   1:  PR[GP1:91,2] = PR[GP1:90,2] + -16.413;
   1:L PR[91] R[100]mm/sec CNT100;
   1:  PR[GP1:91,1] = PR[GP1:90,1] + -9.727;
   1:  PR[GP1:91,2] = PR[GP1:90,2] + -15.652;
   1:L PR[91] R[100]mm/sec CNT100;
   1:  PR[GP1:91,1] = PR[GP1:90,1] + -6.729;
   1:  PR[GP1:91,2] = PR[GP1:90,2] + -12.994;
   1:L PR[91] R[100]mm/sec CNT100;
   1:  PR[GP1:91,1] = PR[GP1:90,1] + -6.347;
   1:  PR[GP1:91,2] = PR[GP1:90,2] + -12.598;
   1:L PR[91] R[100]mm/sec CNT100;
   1:  PR[GP1:91,1] = PR[GP1:90,1] + -4.072;
   1:  PR[GP1:91,2] = PR[GP1:90,2] + -9.212;
   1:L PR[91] R[100]mm/sec CNT100;
   1:  PR[GP1:91,1] = PR[GP1:90,1] + -3.579;
   1:  PR[GP1:91,2] = PR[GP1:90,2] + -8.510;
   1:L PR[91] R[100]mm/sec CNT100;
   1:  PR[GP1:91,1] = PR[GP1:90,1] + -3.207;
   1:  PR[GP1:91,2] = PR[GP1:90,2] + -8.109;
   1:L PR[91] R[100]mm/sec CNT100;
   1:  PR[GP1:91,1] = PR[GP1:90,1] + -2.834;
   1:  PR[GP1:91,2] = PR[GP1:90,2] + -7.762;
   1:L PR[91] R[100]mm/sec CNT100;
   1:  PR[GP1:91,1] = PR[GP1:90,1] + -2.234;
   1:  PR[GP1:91,2] = PR[GP1:90,2] + -7.336;
   1:L PR[91] R[100]mm/sec CNT100;
   1:  PR[GP1:91,1] = PR[GP1:90,1] + -1.110;
   1:  PR[GP1:91,2] = PR[GP1:90,2] + -7.075;
   1:L PR[91] R[100]mm/sec CNT100;
   1:  PR[GP1:91,1] = PR[GP1:90,1] + 1.269;
   1:L PR[91] R[100]mm/sec CNT100;
   1:  PR[GP1:91,1] = PR[GP1:90,1] + 2.391;
   1:  PR[GP1:91,2] = PR[GP1:90,2] + -7.335;
   1:L PR[91] R[100]mm/sec CNT100;
   1:  PR[GP1:91,1] = PR[GP1:90,1] + 2.990;
   1:  PR[GP1:91,2] = PR[GP1:90,2] + -7.760;
   1:L PR[91] R[100]mm/sec CNT100;
   1:  PR[GP1:91,1] = PR[GP1:90,1] + 3.095;
   1:  PR[GP1:91,2] = PR[GP1:90,2] + -7.857;
   1:L PR[91] R[100]mm/sec CNT100;
   1:  PR[GP1:91,1] = PR[GP1:90,1] + 3.258;
   1:  PR[GP1:91,2] = PR[GP1:90,2] + -7.827;
   1:L PR[91] R[100]mm/sec CNT100;
   1:  PR[GP1:91,1] = PR[GP1:90,1] + 4.180;
   1:  PR[GP1:91,2] = PR[GP1:90,2] + -9.139;
   1:L PR[91] R[100]mm/sec CNT100;
   1:  PR[GP1:91,1] = PR[GP1:90,1] + 6.503;
   1:  PR[GP1:91,2] = PR[GP1:90,2] + -12.593;
   1:L PR[91] R[100]mm/sec CNT100;
   1:  PR[GP1:91,1] = PR[GP1:90,1] + 6.887;
   1:  PR[GP1:91,2] = PR[GP1:90,2] + -12.991;
   1:L PR[91] R[100]mm/sec CNT100;
   1:  PR[GP1:91,1] = PR[GP1:90,1] + 9.883;
   1:  PR[GP1:91,2] = PR[GP1:90,2] + -15.654;
   1:L PR[91] R[100]mm/sec CNT100;
   1:  PR[GP1:91,1] = PR[GP1:90,1] + 11.125;
   1:  PR[GP1:91,2] = PR[GP1:90,2] + -16.415;
   1:L PR[91] R[100]mm/sec CNT100;
   1:  PR[GP1:91,1] = PR[GP1:90,1] + 13.931;
   1:  PR[GP1:91,2] = PR[GP1:90,2] + -17.885;
   1:L PR[91] R[100]mm/sec CNT100;
   1:  PR[GP1:91,1] = PR[GP1:90,1] + 16.261;
   1:  PR[GP1:91,2] = PR[GP1:90,2] + -18.611;
   1:L PR[91] R[100]mm/sec CNT100;
   1:  PR[GP1:91,1] = PR[GP1:90,1] + 18.451;
   1:  PR[GP1:91,2] = PR[GP1:90,2] + -19.161;
   1:L PR[91] R[100]mm/sec CNT100;
   1:  PR[GP1:91,1] = PR[GP1:90,1] + 21.839;
   1:  PR[GP1:91,2] = PR[GP1:90,2] + -19.352;
   1:L PR[91] R[100]mm/sec CNT100;
   1:  PR[GP1:91,1] = PR[GP1:90,1] + 23.204;
   1:  PR[GP1:91,2] = PR[GP1:90,2] + -19.363;
   1:L PR[91] R[100]mm/sec CNT100;
   1:  PR[GP1:91,1] = PR[GP1:90,1] + 27.366;
   1:  PR[GP1:91,2] = PR[GP1:90,2] + -18.570;
   1:L PR[91] R[100]mm/sec CNT100;
   1:  PR[GP1:91,1] = PR[GP1:90,1] + 27.918;
   1:  PR[GP1:91,2] = PR[GP1:90,2] + -18.441;
   1:L PR[91] R[100]mm/sec CNT100;
   1:  PR[GP1:91,1] = PR[GP1:90,1] + 32.318;
   1:  PR[GP1:91,2] = PR[GP1:90,2] + -16.403;
   1:L PR[91] R[100]mm/sec CNT100;
   1:  PR[GP1:91,1] = PR[GP1:90,1] + 36.034;
   1:  PR[GP1:91,2] = PR[GP1:90,2] + -13.380;
   1:L PR[91] R[100]mm/sec CNT100;
   1:  PR[GP1:91,1] = PR[GP1:90,1] + 38.885;
   1:  PR[GP1:91,2] = PR[GP1:90,2] + -9.507;
   1:L PR[91] R[100]mm/sec CNT100;
   1:  PR[GP1:91,1] = PR[GP1:90,1] + 40.679;
   1:  PR[GP1:91,2] = PR[GP1:90,2] + -5.092;
   1:L PR[91] R[100]mm/sec CNT100;
   1:  PR[GP1:91,1] = PR[GP1:90,1] + 40.772;
   1:  PR[GP1:91,2] = PR[GP1:90,2] + -4.390;
   1:L PR[91] R[100]mm/sec CNT100;
   1:  PR[GP1:91,1] = PR[GP1:90,1] + 41.290;
   1:  PR[GP1:91,2] = PR[GP1:90,2] + -0.313;
   1:L PR[91] R[100]mm/sec CNT100;
   1:  PR[GP1:91,1] = PR[GP1:90,1] + 40.677;
   1:  PR[GP1:91,2] = PR[GP1:90,2] + 4.471;
   1:L PR[91] R[100]mm/sec CNT100;
   1:  PR[GP1:91,1] = PR[GP1:90,1] + 38.885;
   1:  PR[GP1:91,2] = PR[GP1:90,2] + 8.882;
   1:L PR[91] R[100]mm/sec CNT100;
   1:  PR[GP1:91,1] = PR[GP1:90,1] + 36.035;
   1:  PR[GP1:91,2] = PR[GP1:90,2] + 12.755;
   1:L PR[91] R[100]mm/sec CNT100;
   1:  PR[GP1:91,1] = PR[GP1:90,1] + 32.320;
   1:  PR[GP1:91,2] = PR[GP1:90,2] + 15.778;
   1:L PR[91] R[100]mm/sec CNT100;
   1:  PR[GP1:91,1] = PR[GP1:90,1] + 27.921;
   1:  PR[GP1:91,2] = PR[GP1:90,2] + 17.816;
   1:L PR[91] R[100]mm/sec CNT100;
   1:  PR[GP1:91,1] = PR[GP1:90,1] + 27.368;
   1:  PR[GP1:91,2] = PR[GP1:90,2] + 17.945;
   1:L PR[91] R[100]mm/sec CNT100;
   1:  PR[GP1:91,1] = PR[GP1:90,1] + 23.206;
   1:  PR[GP1:91,2] = PR[GP1:90,2] + 18.739;
   1:L PR[91] R[100]mm/sec CNT100;
   1:  PR[GP1:91,1] = PR[GP1:90,1] + 21.839;
   1:  PR[GP1:91,2] = PR[GP1:90,2] + 18.728;
   1:L PR[91] R[100]mm/sec CNT100;
   1:  PR[GP1:91,1] = PR[GP1:90,1] + 18.450;
   1:  PR[GP1:91,2] = PR[GP1:90,2] + 18.537;
   1:L PR[91] R[100]mm/sec CNT100;
   1:  PR[GP1:91,1] = PR[GP1:90,1] + 16.257;
   1:  PR[GP1:91,2] = PR[GP1:90,2] + 17.986;
   1:L PR[91] R[100]mm/sec CNT100;
   1:  PR[GP1:91,1] = PR[GP1:90,1] + 13.927;
   1:  PR[GP1:91,2] = PR[GP1:90,2] + 17.260;
   1:L PR[91] R[100]mm/sec CNT100;
   1:  PR[GP1:91,1] = PR[GP1:90,1] + 11.119;
   1:  PR[GP1:91,2] = PR[GP1:90,2] + 15.786;
   1:L PR[91] R[100]mm/sec CNT100;
   1:  PR[GP1:91,1] = PR[GP1:90,1] + 9.878;
   1:  PR[GP1:91,2] = PR[GP1:90,2] + 15.026;
   1:L PR[91] R[100]mm/sec CNT100;
   1:  PR[GP1:91,1] = PR[GP1:90,1] + 6.878;
   1:  PR[GP1:91,2] = PR[GP1:90,2] + 12.357;
   1:L PR[91] R[100]mm/sec CNT100;
   1:  PR[GP1:91,1] = PR[GP1:90,1] + 6.495;
   1:  PR[GP1:91,2] = PR[GP1:90,2] + 11.959;
   1:L PR[91] R[100]mm/sec CNT100;
   1:  PR[GP1:91,1] = PR[GP1:90,1] + 3.744;
   1:  PR[GP1:91,2] = PR[GP1:90,2] + 7.889;
   1:L PR[91] R[100]mm/sec CNT100;
   1:  PR[GP1:91,1] = PR[GP1:90,1] + 3.363;
   1:  PR[GP1:91,2] = PR[GP1:90,2] + 7.482;
   1:L PR[91] R[100]mm/sec CNT100;
   1:  PR[GP1:91,1] = PR[GP1:90,1] + 2.992;
   1:  PR[GP1:91,2] = PR[GP1:90,2] + 7.138;
   1:L PR[91] R[100]mm/sec CNT100;
   1:  PR[GP1:91,1] = PR[GP1:90,1] + 2.394;
   1:  PR[GP1:91,2] = PR[GP1:90,2] + 6.712;
   1:L PR[91] R[100]mm/sec CNT100;
   1:  PR[GP1:91,1] = PR[GP1:90,1] + 1.274;
   1:  PR[GP1:91,2] = PR[GP1:90,2] + 6.451;
   1:L PR[91] R[100]mm/sec CNT100;
   1:  PR[GP1:91,1] = PR[GP1:90,1] + -1.109;
   1:L PR[91] R[100]mm/sec CNT100;
   1:  ! -- Layer/Ebene 29 -- !;
   1:  PR[91] = PR[90];
   1:  PR[GP1:91,1] = PR[GP1:90,1] + -2.164;
   1:  PR[GP1:91,2] = PR[GP1:90,2] + 7.007;
   1:  PR[GP1:91,3] = PR[GP1:90,3] + 17.995;
   1:L PR[91] R[100]mm/sec CNT100;
   1:  PR[GP1:91,1] = PR[GP1:90,1] + -2.721;
   1:  PR[GP1:91,2] = PR[GP1:90,2] + 7.403;
   1:L PR[91] R[100]mm/sec CNT100;
   1:  PR[GP1:91,1] = PR[GP1:90,1] + -3.141;
   1:  PR[GP1:91,2] = PR[GP1:90,2] + 7.794;
   1:L PR[91] R[100]mm/sec CNT100;
   1:  PR[GP1:91,1] = PR[GP1:90,1] + -3.471;
   1:  PR[GP1:91,2] = PR[GP1:90,2] + 8.153;
   1:L PR[91] R[100]mm/sec CNT100;
   1:  PR[GP1:91,1] = PR[GP1:90,1] + -6.256;
   1:  PR[GP1:91,2] = PR[GP1:90,2] + 12.114;
   1:L PR[91] R[100]mm/sec CNT100;
   1:  PR[GP1:91,1] = PR[GP1:90,1] + -9.715;
   1:  PR[GP1:91,2] = PR[GP1:90,2] + 15.175;
   1:L PR[91] R[100]mm/sec CNT100;
   1:  PR[GP1:91,1] = PR[GP1:90,1] + -10.311;
   1:  PR[GP1:91,2] = PR[GP1:90,2] + 15.540;
   1:L PR[91] R[100]mm/sec CNT100;
   1:  PR[GP1:91,1] = PR[GP1:90,1] + -13.770;
   1:  PR[GP1:91,2] = PR[GP1:90,2] + 17.357;
   1:L PR[91] R[100]mm/sec CNT100;
   1:  PR[GP1:91,1] = PR[GP1:90,1] + -15.408;
   1:  PR[GP1:91,2] = PR[GP1:90,2] + 17.867;
   1:L PR[91] R[100]mm/sec CNT100;
   1:  PR[GP1:91,1] = PR[GP1:90,1] + -18.283;
   1:  PR[GP1:91,2] = PR[GP1:90,2] + 18.587;
   1:L PR[91] R[100]mm/sec CNT100;
   1:  PR[GP1:91,1] = PR[GP1:90,1] + -20.988;
   1:  PR[GP1:91,2] = PR[GP1:90,2] + 18.739;
   1:L PR[91] R[100]mm/sec CNT100;
   1:  PR[GP1:91,1] = PR[GP1:90,1] + -23.021;
   1:  PR[GP1:91,2] = PR[GP1:90,2] + 18.755;
   1:L PR[91] R[100]mm/sec CNT100;
   1:  PR[GP1:91,1] = PR[GP1:90,1] + -26.552;
   1:  PR[GP1:91,2] = PR[GP1:90,2] + 18.083;
   1:L PR[91] R[100]mm/sec CNT100;
   1:  PR[GP1:91,1] = PR[GP1:90,1] + -27.715;
   1:  PR[GP1:91,2] = PR[GP1:90,2] + 17.812;
   1:L PR[91] R[100]mm/sec CNT100;
   1:  PR[GP1:91,1] = PR[GP1:90,1] + -31.631;
   1:  PR[GP1:91,2] = PR[GP1:90,2] + 15.998;
   1:L PR[91] R[100]mm/sec CNT100;
   1:  PR[GP1:91,1] = PR[GP1:90,1] + -32.075;
   1:  PR[GP1:91,2] = PR[GP1:90,2] + 15.774;
   1:L PR[91] R[100]mm/sec CNT100;
   1:  PR[GP1:91,1] = PR[GP1:90,1] + -35.827;
   1:  PR[GP1:91,2] = PR[GP1:90,2] + 12.731;
   1:L PR[91] R[100]mm/sec CNT100;
   1:  PR[GP1:91,1] = PR[GP1:90,1] + -38.675;
   1:  PR[GP1:91,2] = PR[GP1:90,2] + 8.865;
   1:L PR[91] R[100]mm/sec CNT100;
   1:  PR[GP1:91,1] = PR[GP1:90,1] + -40.458;
   1:  PR[GP1:91,2] = PR[GP1:90,2] + 4.452;
   1:L PR[91] R[100]mm/sec CNT100;
   1:  PR[GP1:91,1] = PR[GP1:90,1] + -41.066;
   1:  PR[GP1:91,2] = PR[GP1:90,2] + -0.312;
   1:L PR[91] R[100]mm/sec CNT100;
   1:  PR[GP1:91,1] = PR[GP1:90,1] + -40.458;
   1:  PR[GP1:91,2] = PR[GP1:90,2] + -5.076;
   1:L PR[91] R[100]mm/sec CNT100;
   1:  PR[GP1:91,1] = PR[GP1:90,1] + -38.674;
   1:  PR[GP1:91,2] = PR[GP1:90,2] + -9.491;
   1:L PR[91] R[100]mm/sec CNT100;
   1:  PR[GP1:91,1] = PR[GP1:90,1] + -36.976;
   1:  PR[GP1:91,2] = PR[GP1:90,2] + -11.803;
   1:L PR[91] R[100]mm/sec CNT100;
   1:  PR[GP1:91,1] = PR[GP1:90,1] + -35.828;
   1:  PR[GP1:91,2] = PR[GP1:90,2] + -13.354;
   1:L PR[91] R[100]mm/sec CNT100;
   1:  PR[GP1:91,1] = PR[GP1:90,1] + -32.074;
   1:  PR[GP1:91,2] = PR[GP1:90,2] + -16.398;
   1:L PR[91] R[100]mm/sec CNT100;
   1:  PR[GP1:91,1] = PR[GP1:90,1] + -31.630;
   1:  PR[GP1:91,2] = PR[GP1:90,2] + -16.622;
   1:L PR[91] R[100]mm/sec CNT100;
   1:  PR[GP1:91,1] = PR[GP1:90,1] + -27.714;
   1:  PR[GP1:91,2] = PR[GP1:90,2] + -18.436;
   1:L PR[91] R[100]mm/sec CNT100;
   1:  PR[GP1:91,1] = PR[GP1:90,1] + -26.551;
   1:  PR[GP1:91,2] = PR[GP1:90,2] + -18.707;
   1:L PR[91] R[100]mm/sec CNT100;
   1:  PR[GP1:91,1] = PR[GP1:90,1] + -23.020;
   1:  PR[GP1:91,2] = PR[GP1:90,2] + -19.379;
   1:L PR[91] R[100]mm/sec CNT100;
   1:  PR[GP1:91,1] = PR[GP1:90,1] + -20.987;
   1:  PR[GP1:91,2] = PR[GP1:90,2] + -19.363;
   1:L PR[91] R[100]mm/sec CNT100;
   1:  PR[GP1:91,1] = PR[GP1:90,1] + -18.282;
   1:  PR[GP1:91,2] = PR[GP1:90,2] + -19.210;
   1:L PR[91] R[100]mm/sec CNT100;
   1:  PR[GP1:91,1] = PR[GP1:90,1] + -15.407;
   1:  PR[GP1:91,2] = PR[GP1:90,2] + -18.491;
   1:L PR[91] R[100]mm/sec CNT100;
   1:  PR[GP1:91,1] = PR[GP1:90,1] + -13.770;
   1:  PR[GP1:91,2] = PR[GP1:90,2] + -17.981;
   1:L PR[91] R[100]mm/sec CNT100;
   1:  PR[GP1:91,1] = PR[GP1:90,1] + -10.310;
   1:  PR[GP1:91,2] = PR[GP1:90,2] + -16.164;
   1:L PR[91] R[100]mm/sec CNT100;
   1:  PR[GP1:91,1] = PR[GP1:90,1] + -9.714;
   1:  PR[GP1:91,2] = PR[GP1:90,2] + -15.798;
   1:L PR[91] R[100]mm/sec CNT100;
   1:  PR[GP1:91,1] = PR[GP1:90,1] + -6.255;
   1:  PR[GP1:91,2] = PR[GP1:90,2] + -12.737;
   1:L PR[91] R[100]mm/sec CNT100;
   1:  PR[GP1:91,1] = PR[GP1:90,1] + -3.471;
   1:  PR[GP1:91,2] = PR[GP1:90,2] + -8.774;
   1:L PR[91] R[100]mm/sec CNT100;
   1:  PR[GP1:91,1] = PR[GP1:90,1] + -3.139;
   1:  PR[GP1:91,2] = PR[GP1:90,2] + -8.415;
   1:L PR[91] R[100]mm/sec CNT100;
   1:  PR[GP1:91,1] = PR[GP1:90,1] + -2.720;
   1:  PR[GP1:91,2] = PR[GP1:90,2] + -8.026;
   1:L PR[91] R[100]mm/sec CNT100;
   1:  PR[GP1:91,1] = PR[GP1:90,1] + -2.163;
   1:  PR[GP1:91,2] = PR[GP1:90,2] + -7.630;
   1:L PR[91] R[100]mm/sec CNT100;
   1:  PR[GP1:91,1] = PR[GP1:90,1] + -1.030;
   1:  PR[GP1:91,2] = PR[GP1:90,2] + -7.363;
   1:L PR[91] R[100]mm/sec CNT100;
   1:  PR[GP1:91,1] = PR[GP1:90,1] + 1.190;
   1:L PR[91] R[100]mm/sec CNT100;
   1:  PR[GP1:91,1] = PR[GP1:90,1] + 2.321;
   1:  PR[GP1:91,2] = PR[GP1:90,2] + -7.630;
   1:L PR[91] R[100]mm/sec CNT100;
   1:  PR[GP1:91,1] = PR[GP1:90,1] + 2.877;
   1:  PR[GP1:91,2] = PR[GP1:90,2] + -8.024;
   1:L PR[91] R[100]mm/sec CNT100;
   1:  PR[GP1:91,1] = PR[GP1:90,1] + 2.984;
   1:  PR[GP1:91,2] = PR[GP1:90,2] + -8.123;
   1:L PR[91] R[100]mm/sec CNT100;
   1:  PR[GP1:91,1] = PR[GP1:90,1] + 3.151;
   1:  PR[GP1:91,2] = PR[GP1:90,2] + -8.091;
   1:L PR[91] R[100]mm/sec CNT100;
   1:  PR[GP1:91,1] = PR[GP1:90,1] + 6.413;
   1:  PR[GP1:91,2] = PR[GP1:90,2] + -12.733;
   1:L PR[91] R[100]mm/sec CNT100;
   1:  PR[GP1:91,1] = PR[GP1:90,1] + 9.871;
   1:  PR[GP1:91,2] = PR[GP1:90,2] + -15.802;
   1:L PR[91] R[100]mm/sec CNT100;
   1:  PR[GP1:91,1] = PR[GP1:90,1] + 10.466;
   1:  PR[GP1:91,2] = PR[GP1:90,2] + -16.166;
   1:L PR[91] R[100]mm/sec CNT100;
   1:  PR[GP1:91,1] = PR[GP1:90,1] + 13.925;
   1:  PR[GP1:91,2] = PR[GP1:90,2] + -17.979;
   1:L PR[91] R[100]mm/sec CNT100;
   1:  PR[GP1:91,1] = PR[GP1:90,1] + 15.563;
   1:  PR[GP1:91,2] = PR[GP1:90,2] + -18.490;
   1:L PR[91] R[100]mm/sec CNT100;
   1:  PR[GP1:91,1] = PR[GP1:90,1] + 18.437;
   1:  PR[GP1:91,2] = PR[GP1:90,2] + -19.210;
   1:L PR[91] R[100]mm/sec CNT100;
   1:  PR[GP1:91,1] = PR[GP1:90,1] + 21.142;
   1:  PR[GP1:91,2] = PR[GP1:90,2] + -19.363;
   1:L PR[91] R[100]mm/sec CNT100;
   1:  PR[GP1:91,1] = PR[GP1:90,1] + 23.175;
   1:  PR[GP1:91,2] = PR[GP1:90,2] + -19.380;
   1:L PR[91] R[100]mm/sec CNT100;
   1:  PR[GP1:91,1] = PR[GP1:90,1] + 26.706;
   1:  PR[GP1:91,2] = PR[GP1:90,2] + -18.707;
   1:L PR[91] R[100]mm/sec CNT100;
   1:  PR[GP1:91,1] = PR[GP1:90,1] + 27.869;
   1:  PR[GP1:91,2] = PR[GP1:90,2] + -18.435;
   1:L PR[91] R[100]mm/sec CNT100;
   1:  PR[GP1:91,1] = PR[GP1:90,1] + 31.786;
   1:  PR[GP1:91,2] = PR[GP1:90,2] + -16.624;
   1:L PR[91] R[100]mm/sec CNT100;
   1:  PR[GP1:91,1] = PR[GP1:90,1] + 32.230;
   1:  PR[GP1:91,2] = PR[GP1:90,2] + -16.401;
   1:L PR[91] R[100]mm/sec CNT100;
   1:  PR[GP1:91,1] = PR[GP1:90,1] + 35.973;
   1:  PR[GP1:91,2] = PR[GP1:90,2] + -13.368;
   1:L PR[91] R[100]mm/sec CNT100;
   1:  PR[GP1:91,1] = PR[GP1:90,1] + 38.831;
   1:  PR[GP1:91,2] = PR[GP1:90,2] + -9.486;
   1:L PR[91] R[100]mm/sec CNT100;
   1:  PR[GP1:91,1] = PR[GP1:90,1] + 40.616;
   1:  PR[GP1:91,2] = PR[GP1:90,2] + -5.083;
   1:L PR[91] R[100]mm/sec CNT100;
   1:  PR[GP1:91,1] = PR[GP1:90,1] + 40.644;
   1:  PR[GP1:91,2] = PR[GP1:90,2] + -4.869;
   1:L PR[91] R[100]mm/sec CNT100;
   1:  PR[GP1:91,1] = PR[GP1:90,1] + 41.223;
   1:  PR[GP1:91,2] = PR[GP1:90,2] + -0.312;
   1:L PR[91] R[100]mm/sec CNT100;
   1:  PR[GP1:91,1] = PR[GP1:90,1] + 40.615;
   1:  PR[GP1:91,2] = PR[GP1:90,2] + 4.462;
   1:L PR[91] R[100]mm/sec CNT100;
   1:  PR[GP1:91,1] = PR[GP1:90,1] + 38.832;
   1:  PR[GP1:91,2] = PR[GP1:90,2] + 8.861;
   1:L PR[91] R[100]mm/sec CNT100;
   1:  PR[GP1:91,1] = PR[GP1:90,1] + 35.983;
   1:  PR[GP1:91,2] = PR[GP1:90,2] + 12.731;
   1:L PR[91] R[100]mm/sec CNT100;
   1:  PR[GP1:91,1] = PR[GP1:90,1] + 32.232;
   1:  PR[GP1:91,2] = PR[GP1:90,2] + 15.776;
   1:L PR[91] R[100]mm/sec CNT100;
   1:  PR[GP1:91,1] = PR[GP1:90,1] + 31.788;
   1:  PR[GP1:91,2] = PR[GP1:90,2] + 15.999;
   1:L PR[91] R[100]mm/sec CNT100;
   1:  PR[GP1:91,1] = PR[GP1:90,1] + 27.870;
   1:  PR[GP1:91,2] = PR[GP1:90,2] + 17.811;
   1:L PR[91] R[100]mm/sec CNT100;
   1:  PR[GP1:91,1] = PR[GP1:90,1] + 26.706;
   1:  PR[GP1:91,2] = PR[GP1:90,2] + 18.082;
   1:L PR[91] R[100]mm/sec CNT100;
   1:  PR[GP1:91,1] = PR[GP1:90,1] + 23.175;
   1:  PR[GP1:91,2] = PR[GP1:90,2] + 18.756;
   1:L PR[91] R[100]mm/sec CNT100;
   1:  PR[GP1:91,1] = PR[GP1:90,1] + 21.139;
   1:  PR[GP1:91,2] = PR[GP1:90,2] + 18.738;
   1:L PR[91] R[100]mm/sec CNT100;
   1:  PR[GP1:91,1] = PR[GP1:90,1] + 18.435;
   1:  PR[GP1:91,2] = PR[GP1:90,2] + 18.586;
   1:L PR[91] R[100]mm/sec CNT100;
   1:  PR[GP1:91,1] = PR[GP1:90,1] + 15.557;
   1:  PR[GP1:91,2] = PR[GP1:90,2] + 17.863;
   1:L PR[91] R[100]mm/sec CNT100;
   1:  PR[GP1:91,1] = PR[GP1:90,1] + 13.919;
   1:  PR[GP1:91,2] = PR[GP1:90,2] + 17.353;
   1:L PR[91] R[100]mm/sec CNT100;
   1:  PR[GP1:91,1] = PR[GP1:90,1] + 10.457;
   1:  PR[GP1:91,2] = PR[GP1:90,2] + 15.535;
   1:L PR[91] R[100]mm/sec CNT100;
   1:  PR[GP1:91,1] = PR[GP1:90,1] + 9.863;
   1:  PR[GP1:91,2] = PR[GP1:90,2] + 15.172;
   1:L PR[91] R[100]mm/sec CNT100;
   1:  PR[GP1:91,1] = PR[GP1:90,1] + 6.404;
   1:  PR[GP1:91,2] = PR[GP1:90,2] + 12.099;
   1:L PR[91] R[100]mm/sec CNT100;
   1:  PR[GP1:91,1] = PR[GP1:90,1] + 3.629;
   1:  PR[GP1:91,2] = PR[GP1:90,2] + 8.144;
   1:L PR[91] R[100]mm/sec CNT100;
   1:  PR[GP1:91,1] = PR[GP1:90,1] + 3.295;
   1:  PR[GP1:91,2] = PR[GP1:90,2] + 7.788;
   1:L PR[91] R[100]mm/sec CNT100;
   1:  PR[GP1:91,1] = PR[GP1:90,1] + 2.879;
   1:  PR[GP1:91,2] = PR[GP1:90,2] + 7.402;
   1:L PR[91] R[100]mm/sec CNT100;
   1:  PR[GP1:91,1] = PR[GP1:90,1] + 2.324;
   1:  PR[GP1:91,2] = PR[GP1:90,2] + 7.007;
   1:L PR[91] R[100]mm/sec CNT100;
   1:  PR[GP1:91,1] = PR[GP1:90,1] + 1.195;
   1:  PR[GP1:91,2] = PR[GP1:90,2] + 6.739;
   1:L PR[91] R[100]mm/sec CNT100;
   1:  PR[GP1:91,1] = PR[GP1:90,1] + -1.030;
   1:L PR[91] R[100]mm/sec CNT100;
   1:  ! -- Layer/Ebene 30 -- !;
   1:  PR[91] = PR[90];
   1:  PR[GP1:91,1] = PR[GP1:90,1] + -2.093;
   1:  PR[GP1:91,2] = PR[GP1:90,2] + 7.301;
   1:  PR[GP1:91,3] = PR[GP1:90,3] + 18.605;
   1:L PR[91] R[100]mm/sec CNT100;
   1:  PR[GP1:91,1] = PR[GP1:90,1] + -2.607;
   1:  PR[GP1:91,2] = PR[GP1:90,2] + 7.667;
   1:L PR[91] R[100]mm/sec CNT100;
   1:  PR[GP1:91,1] = PR[GP1:90,1] + -3.073;
   1:  PR[GP1:91,2] = PR[GP1:90,2] + 8.100;
   1:L PR[91] R[100]mm/sec CNT100;
   1:  PR[GP1:91,1] = PR[GP1:90,1] + -3.365;
   1:  PR[GP1:91,2] = PR[GP1:90,2] + 8.417;
   1:L PR[91] R[100]mm/sec CNT100;
   1:  PR[GP1:91,1] = PR[GP1:90,1] + -5.728;
   1:  PR[GP1:91,2] = PR[GP1:90,2] + 11.782;
   1:L PR[91] R[100]mm/sec CNT100;
   1:  PR[GP1:91,1] = PR[GP1:90,1] + -5.998;
   1:  PR[GP1:91,2] = PR[GP1:90,2] + 12.131;
   1:L PR[91] R[100]mm/sec CNT100;
   1:  PR[GP1:91,1] = PR[GP1:90,1] + -9.684;
   1:  PR[GP1:91,2] = PR[GP1:90,2] + 15.308;
   1:L PR[91] R[100]mm/sec CNT100;
   1:  PR[GP1:91,1] = PR[GP1:90,1] + -13.764;
   1:  PR[GP1:91,2] = PR[GP1:90,2] + 17.451;
   1:L PR[91] R[100]mm/sec CNT100;
   1:  PR[GP1:91,1] = PR[GP1:90,1] + -14.709;
   1:  PR[GP1:91,2] = PR[GP1:90,2] + 17.746;
   1:L PR[91] R[100]mm/sec CNT100;
   1:  PR[GP1:91,1] = PR[GP1:90,1] + -18.269;
   1:  PR[GP1:91,2] = PR[GP1:90,2] + 18.636;
   1:L PR[91] R[100]mm/sec CNT100;
   1:  PR[GP1:91,1] = PR[GP1:90,1] + -20.290;
   1:  PR[GP1:91,2] = PR[GP1:90,2] + 18.750;
   1:L PR[91] R[100]mm/sec CNT100;
   1:  PR[GP1:91,1] = PR[GP1:90,1] + -22.991;
   1:  PR[GP1:91,2] = PR[GP1:90,2] + 18.772;
   1:L PR[91] R[100]mm/sec CNT100;
   1:  PR[GP1:91,1] = PR[GP1:90,1] + -25.892;
   1:  PR[GP1:91,2] = PR[GP1:90,2] + 18.219;
   1:L PR[91] R[100]mm/sec CNT100;
   1:  PR[GP1:91,1] = PR[GP1:90,1] + -27.664;
   1:  PR[GP1:91,2] = PR[GP1:90,2] + 17.807;
   1:L PR[91] R[100]mm/sec CNT100;
   1:  PR[GP1:91,1] = PR[GP1:90,1] + -31.036;
   1:  PR[GP1:91,2] = PR[GP1:90,2] + 16.244;
   1:L PR[91] R[100]mm/sec CNT100;
   1:  PR[GP1:91,1] = PR[GP1:90,1] + -32.004;
   1:  PR[GP1:91,2] = PR[GP1:90,2] + 15.757;
   1:L PR[91] R[100]mm/sec CNT100;
   1:  PR[GP1:91,1] = PR[GP1:90,1] + -35.336;
   1:  PR[GP1:91,2] = PR[GP1:90,2] + 13.058;
   1:L PR[91] R[100]mm/sec CNT100;
   1:  PR[GP1:91,1] = PR[GP1:90,1] + -35.728;
   1:  PR[GP1:91,2] = PR[GP1:90,2] + 12.724;
   1:L PR[91] R[100]mm/sec CNT100;
   1:  PR[GP1:91,1] = PR[GP1:90,1] + -38.512;
   1:  PR[GP1:91,2] = PR[GP1:90,2] + 8.963;
   1:L PR[91] R[100]mm/sec CNT100;
   1:  PR[GP1:91,1] = PR[GP1:90,1] + -38.587;
   1:  PR[GP1:91,2] = PR[GP1:90,2] + 8.857;
   1:L PR[91] R[100]mm/sec CNT100;
   1:  PR[GP1:91,1] = PR[GP1:90,1] + -40.387;
   1:  PR[GP1:91,2] = PR[GP1:90,2] + 4.439;
   1:L PR[91] R[100]mm/sec CNT100;
   1:  PR[GP1:91,1] = PR[GP1:90,1] + -41.000;
   1:  PR[GP1:91,2] = PR[GP1:90,2] + -0.312;
   1:L PR[91] R[100]mm/sec CNT100;
   1:  PR[GP1:91,1] = PR[GP1:90,1] + -40.387;
   1:  PR[GP1:91,2] = PR[GP1:90,2] + -5.063;
   1:L PR[91] R[100]mm/sec CNT100;
   1:  PR[GP1:91,1] = PR[GP1:90,1] + -38.592;
   1:  PR[GP1:91,2] = PR[GP1:90,2] + -9.468;
   1:L PR[91] R[100]mm/sec CNT100;
   1:  PR[GP1:91,1] = PR[GP1:90,1] + -35.727;
   1:  PR[GP1:91,2] = PR[GP1:90,2] + -13.349;
   1:L PR[91] R[100]mm/sec CNT100;
   1:  PR[GP1:91,1] = PR[GP1:90,1] + -35.335;
   1:  PR[GP1:91,2] = PR[GP1:90,2] + -13.683;
   1:L PR[91] R[100]mm/sec CNT100;
   1:  PR[GP1:91,1] = PR[GP1:90,1] + -32.004;
   1:  PR[GP1:91,2] = PR[GP1:90,2] + -16.381;
   1:L PR[91] R[100]mm/sec CNT100;
   1:  PR[GP1:91,1] = PR[GP1:90,1] + -31.036;
   1:  PR[GP1:91,2] = PR[GP1:90,2] + -16.869;
   1:L PR[91] R[100]mm/sec CNT100;
   1:  PR[GP1:91,1] = PR[GP1:90,1] + -27.664;
   1:  PR[GP1:91,2] = PR[GP1:90,2] + -18.431;
   1:L PR[91] R[100]mm/sec CNT100;
   1:  PR[GP1:91,1] = PR[GP1:90,1] + -25.891;
   1:  PR[GP1:91,2] = PR[GP1:90,2] + -18.843;
   1:L PR[91] R[100]mm/sec CNT100;
   1:  PR[GP1:91,1] = PR[GP1:90,1] + -22.990;
   1:  PR[GP1:91,2] = PR[GP1:90,2] + -19.396;
   1:L PR[91] R[100]mm/sec CNT100;
   1:  PR[GP1:91,1] = PR[GP1:90,1] + -20.289;
   1:  PR[GP1:91,2] = PR[GP1:90,2] + -19.374;
   1:L PR[91] R[100]mm/sec CNT100;
   1:  PR[GP1:91,1] = PR[GP1:90,1] + -18.268;
   1:  PR[GP1:91,2] = PR[GP1:90,2] + -19.260;
   1:L PR[91] R[100]mm/sec CNT100;
   1:  PR[GP1:91,1] = PR[GP1:90,1] + -14.708;
   1:  PR[GP1:91,2] = PR[GP1:90,2] + -18.369;
   1:L PR[91] R[100]mm/sec CNT100;
   1:  PR[GP1:91,1] = PR[GP1:90,1] + -13.763;
   1:  PR[GP1:91,2] = PR[GP1:90,2] + -18.075;
   1:L PR[91] R[100]mm/sec CNT100;
   1:  PR[GP1:91,1] = PR[GP1:90,1] + -9.690;
   1:  PR[GP1:91,2] = PR[GP1:90,2] + -15.935;
   1:L PR[91] R[100]mm/sec CNT100;
   1:  PR[GP1:91,1] = PR[GP1:90,1] + -9.338;
   1:  PR[GP1:91,2] = PR[GP1:90,2] + -15.623;
   1:L PR[91] R[100]mm/sec CNT100;
   1:  PR[GP1:91,1] = PR[GP1:90,1] + -6.247;
   1:  PR[GP1:91,2] = PR[GP1:90,2] + -12.988;
   1:L PR[91] R[100]mm/sec CNT100;
   1:  PR[GP1:91,1] = PR[GP1:90,1] + -6.011;
   1:  PR[GP1:91,2] = PR[GP1:90,2] + -12.772;
   1:L PR[91] R[100]mm/sec CNT100;
   1:  PR[GP1:91,1] = PR[GP1:90,1] + -5.728;
   1:  PR[GP1:91,2] = PR[GP1:90,2] + -12.406;
   1:L PR[91] R[100]mm/sec CNT100;
   1:  PR[GP1:91,1] = PR[GP1:90,1] + -3.364;
   1:  PR[GP1:91,2] = PR[GP1:90,2] + -9.038;
   1:L PR[91] R[100]mm/sec CNT100;
   1:  PR[GP1:91,1] = PR[GP1:90,1] + -3.070;
   1:  PR[GP1:91,2] = PR[GP1:90,2] + -8.722;
   1:L PR[91] R[100]mm/sec CNT100;
   1:  PR[GP1:91,1] = PR[GP1:90,1] + -2.607;
   1:  PR[GP1:91,2] = PR[GP1:90,2] + -8.291;
   1:L PR[91] R[100]mm/sec CNT100;
   1:  PR[GP1:91,1] = PR[GP1:90,1] + -2.093;
   1:  PR[GP1:91,2] = PR[GP1:90,2] + -7.925;
   1:L PR[91] R[100]mm/sec CNT100;
   1:  PR[GP1:91,1] = PR[GP1:90,1] + -0.950;
   1:  PR[GP1:91,2] = PR[GP1:90,2] + -7.652;
   1:L PR[91] R[100]mm/sec CNT100;
   1:  PR[GP1:91,1] = PR[GP1:90,1] + 1.111;
   1:L PR[91] R[100]mm/sec CNT100;
   1:  PR[GP1:91,1] = PR[GP1:90,1] + 2.251;
   1:  PR[GP1:91,2] = PR[GP1:90,2] + -7.924;
   1:L PR[91] R[100]mm/sec CNT100;
   1:  PR[GP1:91,1] = PR[GP1:90,1] + 2.765;
   1:  PR[GP1:91,2] = PR[GP1:90,2] + -8.288;
   1:L PR[91] R[100]mm/sec CNT100;
   1:  PR[GP1:91,1] = PR[GP1:90,1] + 2.872;
   1:  PR[GP1:91,2] = PR[GP1:90,2] + -8.388;
   1:L PR[91] R[100]mm/sec CNT100;
   1:  PR[GP1:91,1] = PR[GP1:90,1] + 3.046;
   1:  PR[GP1:91,2] = PR[GP1:90,2] + -8.355;
   1:L PR[91] R[100]mm/sec CNT100;
   1:  PR[GP1:91,1] = PR[GP1:90,1] + 5.886;
   1:  PR[GP1:91,2] = PR[GP1:90,2] + -12.401;
   1:L PR[91] R[100]mm/sec CNT100;
   1:  PR[GP1:91,1] = PR[GP1:90,1] + 6.159;
   1:  PR[GP1:91,2] = PR[GP1:90,2] + -12.754;
   1:L PR[91] R[100]mm/sec CNT100;
   1:  PR[GP1:91,1] = PR[GP1:90,1] + 9.840;
   1:  PR[GP1:91,2] = PR[GP1:90,2] + -15.935;
   1:L PR[91] R[100]mm/sec CNT100;
   1:  PR[GP1:91,1] = PR[GP1:90,1] + 13.919;
   1:  PR[GP1:91,2] = PR[GP1:90,2] + -18.073;
   1:L PR[91] R[100]mm/sec CNT100;
   1:  PR[GP1:91,1] = PR[GP1:90,1] + 14.865;
   1:  PR[GP1:91,2] = PR[GP1:90,2] + -18.368;
   1:L PR[91] R[100]mm/sec CNT100;
   1:  PR[GP1:91,1] = PR[GP1:90,1] + 18.424;
   1:  PR[GP1:91,2] = PR[GP1:90,2] + -19.260;
   1:L PR[91] R[100]mm/sec CNT100;
   1:  PR[GP1:91,1] = PR[GP1:90,1] + 20.445;
   1:  PR[GP1:91,2] = PR[GP1:90,2] + -19.374;
   1:L PR[91] R[100]mm/sec CNT100;
   1:  PR[GP1:91,1] = PR[GP1:90,1] + 23.145;
   1:  PR[GP1:91,2] = PR[GP1:90,2] + -19.396;
   1:L PR[91] R[100]mm/sec CNT100;
   1:  PR[GP1:91,1] = PR[GP1:90,1] + 26.046;
   1:  PR[GP1:91,2] = PR[GP1:90,2] + -18.843;
   1:L PR[91] R[100]mm/sec CNT100;
   1:  PR[GP1:91,1] = PR[GP1:90,1] + 27.819;
   1:  PR[GP1:91,2] = PR[GP1:90,2] + -18.430;
   1:L PR[91] R[100]mm/sec CNT100;
   1:  PR[GP1:91,1] = PR[GP1:90,1] + 31.192;
   1:  PR[GP1:91,2] = PR[GP1:90,2] + -16.870;
   1:L PR[91] R[100]mm/sec CNT100;
   1:  PR[GP1:91,1] = PR[GP1:90,1] + 32.160;
   1:  PR[GP1:91,2] = PR[GP1:90,2] + -16.383;
   1:L PR[91] R[100]mm/sec CNT100;
   1:  PR[GP1:91,1] = PR[GP1:90,1] + 35.491;
   1:  PR[GP1:91,2] = PR[GP1:90,2] + -13.684;
   1:L PR[91] R[100]mm/sec CNT100;
   1:  PR[GP1:91,1] = PR[GP1:90,1] + 35.883;
   1:  PR[GP1:91,2] = PR[GP1:90,2] + -13.349;
   1:L PR[91] R[100]mm/sec CNT100;
   1:  PR[GP1:91,1] = PR[GP1:90,1] + 38.667;
   1:  PR[GP1:91,2] = PR[GP1:90,2] + -9.585;
   1:L PR[91] R[100]mm/sec CNT100;
   1:  PR[GP1:91,1] = PR[GP1:90,1] + 38.744;
   1:  PR[GP1:91,2] = PR[GP1:90,2] + -9.477;
   1:L PR[91] R[100]mm/sec CNT100;
   1:  PR[GP1:91,1] = PR[GP1:90,1] + 40.543;
   1:  PR[GP1:91,2] = PR[GP1:90,2] + -5.075;
   1:L PR[91] R[100]mm/sec CNT100;
   1:  PR[GP1:91,1] = PR[GP1:90,1] + 41.157;
   1:  PR[GP1:91,2] = PR[GP1:90,2] + -0.312;
   1:L PR[91] R[100]mm/sec CNT100;
   1:  PR[GP1:91,1] = PR[GP1:90,1] + 40.543;
   1:  PR[GP1:91,2] = PR[GP1:90,2] + 4.450;
   1:L PR[91] R[100]mm/sec CNT100;
   1:  PR[GP1:91,1] = PR[GP1:90,1] + 38.749;
   1:  PR[GP1:91,2] = PR[GP1:90,2] + 8.839;
   1:L PR[91] R[100]mm/sec CNT100;
   1:  PR[GP1:91,1] = PR[GP1:90,1] + 35.883;
   1:  PR[GP1:91,2] = PR[GP1:90,2] + 12.725;
   1:L PR[91] R[100]mm/sec CNT100;
   1:  PR[GP1:91,1] = PR[GP1:90,1] + 35.492;
   1:  PR[GP1:91,2] = PR[GP1:90,2] + 13.059;
   1:L PR[91] R[100]mm/sec CNT100;
   1:  PR[GP1:91,1] = PR[GP1:90,1] + 32.161;
   1:  PR[GP1:91,2] = PR[GP1:90,2] + 15.759;
   1:L PR[91] R[100]mm/sec CNT100;
   1:  PR[GP1:91,1] = PR[GP1:90,1] + 31.192;
   1:  PR[GP1:91,2] = PR[GP1:90,2] + 16.245;
   1:L PR[91] R[100]mm/sec CNT100;
   1:  PR[GP1:91,1] = PR[GP1:90,1] + 27.819;
   1:  PR[GP1:91,2] = PR[GP1:90,2] + 17.806;
   1:L PR[91] R[100]mm/sec CNT100;
   1:  PR[GP1:91,1] = PR[GP1:90,1] + 26.044;
   1:  PR[GP1:91,2] = PR[GP1:90,2] + 18.219;
   1:L PR[91] R[100]mm/sec CNT100;
   1:  PR[GP1:91,1] = PR[GP1:90,1] + 23.144;
   1:  PR[GP1:91,2] = PR[GP1:90,2] + 18.773;
   1:L PR[91] R[100]mm/sec CNT100;
   1:  PR[GP1:91,1] = PR[GP1:90,1] + 20.440;
   1:  PR[GP1:91,2] = PR[GP1:90,2] + 18.749;
   1:L PR[91] R[100]mm/sec CNT100;
   1:  PR[GP1:91,1] = PR[GP1:90,1] + 18.419;
   1:  PR[GP1:91,2] = PR[GP1:90,2] + 18.636;
   1:L PR[91] R[100]mm/sec CNT100;
   1:  PR[GP1:91,1] = PR[GP1:90,1] + 14.856;
   1:  PR[GP1:91,2] = PR[GP1:90,2] + 17.741;
   1:L PR[91] R[100]mm/sec CNT100;
   1:  PR[GP1:91,1] = PR[GP1:90,1] + 13.913;
   1:  PR[GP1:91,2] = PR[GP1:90,2] + 17.447;
   1:L PR[91] R[100]mm/sec CNT100;
   1:  PR[GP1:91,1] = PR[GP1:90,1] + 9.816;
   1:  PR[GP1:91,2] = PR[GP1:90,2] + 15.288;
   1:L PR[91] R[100]mm/sec CNT100;
   1:  PR[GP1:91,1] = PR[GP1:90,1] + 9.497;
   1:  PR[GP1:91,2] = PR[GP1:90,2] + 15.005;
   1:L PR[91] R[100]mm/sec CNT100;
   1:  PR[GP1:91,1] = PR[GP1:90,1] + 6.399;
   1:  PR[GP1:91,2] = PR[GP1:90,2] + 12.354;
   1:L PR[91] R[100]mm/sec CNT100;
   1:  PR[GP1:91,1] = PR[GP1:90,1] + 6.164;
   1:  PR[GP1:91,2] = PR[GP1:90,2] + 12.138;
   1:L PR[91] R[100]mm/sec CNT100;
   1:  PR[GP1:91,1] = PR[GP1:90,1] + 5.877;
   1:  PR[GP1:91,2] = PR[GP1:90,2] + 11.767;
   1:L PR[91] R[100]mm/sec CNT100;
   1:  PR[GP1:91,1] = PR[GP1:90,1] + 3.522;
   1:  PR[GP1:91,2] = PR[GP1:90,2] + 8.409;
   1:L PR[91] R[100]mm/sec CNT100;
   1:  PR[GP1:91,1] = PR[GP1:90,1] + 3.228;
   1:  PR[GP1:91,2] = PR[GP1:90,2] + 8.094;
   1:L PR[91] R[100]mm/sec CNT100;
   1:  PR[GP1:91,1] = PR[GP1:90,1] + 2.767;
   1:  PR[GP1:91,2] = PR[GP1:90,2] + 7.666;
   1:L PR[91] R[100]mm/sec CNT100;
   1:  PR[GP1:91,1] = PR[GP1:90,1] + 2.254;
   1:  PR[GP1:91,2] = PR[GP1:90,2] + 7.301;
   1:L PR[91] R[100]mm/sec CNT100;
   1:  PR[GP1:91,1] = PR[GP1:90,1] + 1.115;
   1:  PR[GP1:91,2] = PR[GP1:90,2] + 7.028;
   1:L PR[91] R[100]mm/sec CNT100;
   1:  PR[GP1:91,1] = PR[GP1:90,1] + -0.950;
   1:L PR[91] R[100]mm/sec CNT100;
   1:  ! -- Layer/Ebene 31 -- !;
   1:  PR[91] = PR[90];
   1:  PR[GP1:91,1] = PR[GP1:90,1] + -2.023;
   1:  PR[GP1:91,2] = PR[GP1:90,2] + 7.596;
   1:  PR[GP1:91,3] = PR[GP1:90,3] + 19.215;
   1:L PR[91] R[100]mm/sec CNT100;
   1:  PR[GP1:91,1] = PR[GP1:90,1] + -2.494;
   1:  PR[GP1:91,2] = PR[GP1:90,2] + 7.931;
   1:L PR[91] R[100]mm/sec CNT100;
   1:  PR[GP1:91,1] = PR[GP1:90,1] + -3.005;
   1:  PR[GP1:91,2] = PR[GP1:90,2] + 8.406;
   1:L PR[91] R[100]mm/sec CNT100;
   1:  PR[GP1:91,1] = PR[GP1:90,1] + -3.258;
   1:  PR[GP1:91,2] = PR[GP1:90,2] + 8.681;
   1:L PR[91] R[100]mm/sec CNT100;
   1:  PR[GP1:91,1] = PR[GP1:90,1] + -5.146;
   1:  PR[GP1:91,2] = PR[GP1:90,2] + 11.370;
   1:L PR[91] R[100]mm/sec CNT100;
   1:  PR[GP1:91,1] = PR[GP1:90,1] + -5.771;
   1:  PR[GP1:91,2] = PR[GP1:90,2] + 12.177;
   1:L PR[91] R[100]mm/sec CNT100;
   1:  PR[GP1:91,1] = PR[GP1:90,1] + -9.006;
   1:  PR[GP1:91,2] = PR[GP1:90,2] + 14.955;
   1:L PR[91] R[100]mm/sec CNT100;
   1:  PR[GP1:91,1] = PR[GP1:90,1] + -9.356;
   1:  PR[GP1:91,2] = PR[GP1:90,2] + 15.271;
   1:L PR[91] R[100]mm/sec CNT100;
   1:  PR[GP1:91,1] = PR[GP1:90,1] + -9.540;
   1:  PR[GP1:91,2] = PR[GP1:90,2] + 15.393;
   1:L PR[91] R[100]mm/sec CNT100;
   1:  PR[GP1:91,1] = PR[GP1:90,1] + -12.048;
   1:  PR[GP1:91,2] = PR[GP1:90,2] + 16.647;
   1:L PR[91] R[100]mm/sec CNT100;
   1:  PR[GP1:91,1] = PR[GP1:90,1] + -13.757;
   1:  PR[GP1:91,2] = PR[GP1:90,2] + 17.545;
   1:L PR[91] R[100]mm/sec CNT100;
   1:  PR[GP1:91,1] = PR[GP1:90,1] + -14.011;
   1:  PR[GP1:91,2] = PR[GP1:90,2] + 17.624;
   1:L PR[91] R[100]mm/sec CNT100;
   1:  PR[GP1:91,1] = PR[GP1:90,1] + -18.255;
   1:  PR[GP1:91,2] = PR[GP1:90,2] + 18.686;
   1:L PR[91] R[100]mm/sec CNT100;
   1:  PR[GP1:91,1] = PR[GP1:90,1] + -19.593;
   1:  PR[GP1:91,2] = PR[GP1:90,2] + 18.761;
   1:L PR[91] R[100]mm/sec CNT100;
   1:  PR[GP1:91,1] = PR[GP1:90,1] + -22.960;
   1:  PR[GP1:91,2] = PR[GP1:90,2] + 18.788;
   1:L PR[91] R[100]mm/sec CNT100;
   1:  PR[GP1:91,1] = PR[GP1:90,1] + -25.231;
   1:  PR[GP1:91,2] = PR[GP1:90,2] + 18.356;
   1:L PR[91] R[100]mm/sec CNT100;
   1:  PR[GP1:91,1] = PR[GP1:90,1] + -27.614;
   1:  PR[GP1:91,2] = PR[GP1:90,2] + 17.801;
   1:L PR[91] R[100]mm/sec CNT100;
   1:  PR[GP1:91,1] = PR[GP1:90,1] + -30.442;
   1:  PR[GP1:91,2] = PR[GP1:90,2] + 16.491;
   1:L PR[91] R[100]mm/sec CNT100;
   1:  PR[GP1:91,1] = PR[GP1:90,1] + -31.933;
   1:  PR[GP1:91,2] = PR[GP1:90,2] + 15.740;
   1:L PR[91] R[100]mm/sec CNT100;
   1:  PR[GP1:91,1] = PR[GP1:90,1] + -34.830;
   1:  PR[GP1:91,2] = PR[GP1:90,2] + 13.394;
   1:L PR[91] R[100]mm/sec CNT100;
   1:  PR[GP1:91,1] = PR[GP1:90,1] + -35.638;
   1:  PR[GP1:91,2] = PR[GP1:90,2] + 12.704;
   1:L PR[91] R[100]mm/sec CNT100;
   1:  PR[GP1:91,1] = PR[GP1:90,1] + -38.108;
   1:  PR[GP1:91,2] = PR[GP1:90,2] + 9.367;
   1:L PR[91] R[100]mm/sec CNT100;
   1:  PR[GP1:91,1] = PR[GP1:90,1] + -38.483;
   1:  PR[GP1:91,2] = PR[GP1:90,2] + 8.839;
   1:L PR[91] R[100]mm/sec CNT100;
   1:  PR[GP1:91,1] = PR[GP1:90,1] + -40.274;
   1:  PR[GP1:91,2] = PR[GP1:90,2] + 4.432;
   1:L PR[91] R[100]mm/sec CNT100;
   1:  PR[GP1:91,1] = PR[GP1:90,1] + -40.854;
   1:  PR[GP1:91,2] = PR[GP1:90,2] + -0.064;
   1:L PR[91] R[100]mm/sec CNT100;
   1:  PR[GP1:91,1] = PR[GP1:90,1] + -40.903;
   1:  PR[GP1:91,2] = PR[GP1:90,2] + -0.342;
   1:L PR[91] R[100]mm/sec CNT100;
   1:  PR[GP1:91,1] = PR[GP1:90,1] + -40.274;
   1:  PR[GP1:91,2] = PR[GP1:90,2] + -5.059;
   1:L PR[91] R[100]mm/sec CNT100;
   1:  PR[GP1:91,1] = PR[GP1:90,1] + -40.131;
   1:  PR[GP1:91,2] = PR[GP1:90,2] + -5.419;
   1:L PR[91] R[100]mm/sec CNT100;
   1:  PR[GP1:91,1] = PR[GP1:90,1] + -38.483;
   1:  PR[GP1:91,2] = PR[GP1:90,2] + -9.463;
   1:L PR[91] R[100]mm/sec CNT100;
   1:  PR[GP1:91,1] = PR[GP1:90,1] + -38.108;
   1:  PR[GP1:91,2] = PR[GP1:90,2] + -9.991;
   1:L PR[91] R[100]mm/sec CNT100;
   1:  PR[GP1:91,1] = PR[GP1:90,1] + -35.638;
   1:  PR[GP1:91,2] = PR[GP1:90,2] + -13.329;
   1:L PR[91] R[100]mm/sec CNT100;
   1:  PR[GP1:91,1] = PR[GP1:90,1] + -34.829;
   1:  PR[GP1:91,2] = PR[GP1:90,2] + -14.018;
   1:L PR[91] R[100]mm/sec CNT100;
   1:  PR[GP1:91,1] = PR[GP1:90,1] + -31.933;
   1:  PR[GP1:91,2] = PR[GP1:90,2] + -16.364;
   1:L PR[91] R[100]mm/sec CNT100;
   1:  PR[GP1:91,1] = PR[GP1:90,1] + -30.442;
   1:  PR[GP1:91,2] = PR[GP1:90,2] + -17.115;
   1:L PR[91] R[100]mm/sec CNT100;
   1:  PR[GP1:91,1] = PR[GP1:90,1] + -27.613;
   1:  PR[GP1:91,2] = PR[GP1:90,2] + -18.425;
   1:L PR[91] R[100]mm/sec CNT100;
   1:  PR[GP1:91,1] = PR[GP1:90,1] + -25.230;
   1:  PR[GP1:91,2] = PR[GP1:90,2] + -18.980;
   1:L PR[91] R[100]mm/sec CNT100;
   1:  PR[GP1:91,1] = PR[GP1:90,1] + -22.960;
   1:  PR[GP1:91,2] = PR[GP1:90,2] + -19.413;
   1:L PR[91] R[100]mm/sec CNT100;
   1:  PR[GP1:91,1] = PR[GP1:90,1] + -19.592;
   1:  PR[GP1:91,2] = PR[GP1:90,2] + -19.385;
   1:L PR[91] R[100]mm/sec CNT100;
   1:  PR[GP1:91,1] = PR[GP1:90,1] + -18.254;
   1:  PR[GP1:91,2] = PR[GP1:90,2] + -19.310;
   1:L PR[91] R[100]mm/sec CNT100;
   1:  PR[GP1:91,1] = PR[GP1:90,1] + -14.010;
   1:  PR[GP1:91,2] = PR[GP1:90,2] + -18.248;
   1:L PR[91] R[100]mm/sec CNT100;
   1:  PR[GP1:91,1] = PR[GP1:90,1] + -13.757;
   1:  PR[GP1:91,2] = PR[GP1:90,2] + -18.169;
   1:L PR[91] R[100]mm/sec CNT100;
   1:  PR[GP1:91,1] = PR[GP1:90,1] + -12.048;
   1:  PR[GP1:91,2] = PR[GP1:90,2] + -17.271;
   1:L PR[91] R[100]mm/sec CNT100;
   1:  PR[GP1:91,1] = PR[GP1:90,1] + -9.539;
   1:  PR[GP1:91,2] = PR[GP1:90,2] + -16.017;
   1:L PR[91] R[100]mm/sec CNT100;
   1:  PR[GP1:91,1] = PR[GP1:90,1] + -9.337;
   1:  PR[GP1:91,2] = PR[GP1:90,2] + -15.883;
   1:L PR[91] R[100]mm/sec CNT100;
   1:  PR[GP1:91,1] = PR[GP1:90,1] + -6.343;
   1:  PR[GP1:91,2] = PR[GP1:90,2] + -13.331;
   1:L PR[91] R[100]mm/sec CNT100;
   1:  PR[GP1:91,1] = PR[GP1:90,1] + -5.785;
   1:  PR[GP1:91,2] = PR[GP1:90,2] + -12.819;
   1:L PR[91] R[100]mm/sec CNT100;
   1:  PR[GP1:91,1] = PR[GP1:90,1] + -5.146;
   1:  PR[GP1:91,2] = PR[GP1:90,2] + -11.994;
   1:L PR[91] R[100]mm/sec CNT100;
   1:  PR[GP1:91,1] = PR[GP1:90,1] + -3.257;
   1:  PR[GP1:91,2] = PR[GP1:90,2] + -9.302;
   1:L PR[91] R[100]mm/sec CNT100;
   1:  PR[GP1:91,1] = PR[GP1:90,1] + -3.002;
   1:  PR[GP1:91,2] = PR[GP1:90,2] + -9.028;
   1:L PR[91] R[100]mm/sec CNT100;
   1:  PR[GP1:91,1] = PR[GP1:90,1] + -2.493;
   1:  PR[GP1:91,2] = PR[GP1:90,2] + -8.555;
   1:L PR[91] R[100]mm/sec CNT100;
   1:  PR[GP1:91,1] = PR[GP1:90,1] + -2.022;
   1:  PR[GP1:91,2] = PR[GP1:90,2] + -8.220;
   1:L PR[91] R[100]mm/sec CNT100;
   1:  PR[GP1:91,1] = PR[GP1:90,1] + -0.870;
   1:  PR[GP1:91,2] = PR[GP1:90,2] + -7.940;
   1:L PR[91] R[100]mm/sec CNT100;
   1:  PR[GP1:91,1] = PR[GP1:90,1] + 1.032;
   1:L PR[91] R[100]mm/sec CNT100;
   1:  PR[GP1:91,1] = PR[GP1:90,1] + 2.182;
   1:  PR[GP1:91,2] = PR[GP1:90,2] + -8.219;
   1:L PR[91] R[100]mm/sec CNT100;
   1:  PR[GP1:91,1] = PR[GP1:90,1] + 2.652;
   1:  PR[GP1:91,2] = PR[GP1:90,2] + -8.553;
   1:L PR[91] R[100]mm/sec CNT100;
   1:  PR[GP1:91,1] = PR[GP1:90,1] + 2.761;
   1:  PR[GP1:91,2] = PR[GP1:90,2] + -8.654;
   1:L PR[91] R[100]mm/sec CNT100;
   1:  PR[GP1:91,1] = PR[GP1:90,1] + 2.939;
   1:  PR[GP1:91,2] = PR[GP1:90,2] + -8.620;
   1:L PR[91] R[100]mm/sec CNT100;
   1:  PR[GP1:91,1] = PR[GP1:90,1] + 5.305;
   1:  PR[GP1:91,2] = PR[GP1:90,2] + -11.990;
   1:L PR[91] R[100]mm/sec CNT100;
   1:  PR[GP1:91,1] = PR[GP1:90,1] + 5.936;
   1:  PR[GP1:91,2] = PR[GP1:90,2] + -12.804;
   1:L PR[91] R[100]mm/sec CNT100;
   1:  PR[GP1:91,1] = PR[GP1:90,1] + 9.168;
   1:  PR[GP1:91,2] = PR[GP1:90,2] + -15.586;
   1:L PR[91] R[100]mm/sec CNT100;
   1:  PR[GP1:91,1] = PR[GP1:90,1] + 9.515;
   1:  PR[GP1:91,2] = PR[GP1:90,2] + -15.900;
   1:L PR[91] R[100]mm/sec CNT100;
   1:  PR[GP1:91,1] = PR[GP1:90,1] + 9.695;
   1:  PR[GP1:91,2] = PR[GP1:90,2] + -16.019;
   1:L PR[91] R[100]mm/sec CNT100;
   1:  PR[GP1:91,1] = PR[GP1:90,1] + 12.203;
   1:  PR[GP1:91,2] = PR[GP1:90,2] + -17.271;
   1:L PR[91] R[100]mm/sec CNT100;
   1:  PR[GP1:91,1] = PR[GP1:90,1] + 13.913;
   1:  PR[GP1:91,2] = PR[GP1:90,2] + -18.167;
   1:L PR[91] R[100]mm/sec CNT100;
   1:  PR[GP1:91,1] = PR[GP1:90,1] + 14.167;
   1:  PR[GP1:91,2] = PR[GP1:90,2] + -18.246;
   1:L PR[91] R[100]mm/sec CNT100;
   1:  PR[GP1:91,1] = PR[GP1:90,1] + 18.410;
   1:  PR[GP1:91,2] = PR[GP1:90,2] + -19.310;
   1:L PR[91] R[100]mm/sec CNT100;
   1:  PR[GP1:91,1] = PR[GP1:90,1] + 19.748;
   1:  PR[GP1:91,2] = PR[GP1:90,2] + -19.385;
   1:L PR[91] R[100]mm/sec CNT100;
   1:  PR[GP1:91,1] = PR[GP1:90,1] + 23.115;
   1:  PR[GP1:91,2] = PR[GP1:90,2] + -19.413;
   1:L PR[91] R[100]mm/sec CNT100;
   1:  PR[GP1:91,1] = PR[GP1:90,1] + 25.386;
   1:  PR[GP1:91,2] = PR[GP1:90,2] + -18.980;
   1:L PR[91] R[100]mm/sec CNT100;
   1:  PR[GP1:91,1] = PR[GP1:90,1] + 27.769;
   1:  PR[GP1:91,2] = PR[GP1:90,2] + -18.424;
   1:L PR[91] R[100]mm/sec CNT100;
   1:  PR[GP1:91,1] = PR[GP1:90,1] + 30.598;
   1:  PR[GP1:91,2] = PR[GP1:90,2] + -17.116;
   1:L PR[91] R[100]mm/sec CNT100;
   1:  PR[GP1:91,1] = PR[GP1:90,1] + 32.089;
   1:  PR[GP1:91,2] = PR[GP1:90,2] + -16.366;
   1:L PR[91] R[100]mm/sec CNT100;
   1:  PR[GP1:91,1] = PR[GP1:90,1] + 34.985;
   1:  PR[GP1:91,2] = PR[GP1:90,2] + -14.020;
   1:L PR[91] R[100]mm/sec CNT100;
   1:  PR[GP1:91,1] = PR[GP1:90,1] + 35.793;
   1:  PR[GP1:91,2] = PR[GP1:90,2] + -13.329;
   1:L PR[91] R[100]mm/sec CNT100;
   1:  PR[GP1:91,1] = PR[GP1:90,1] + 38.264;
   1:  PR[GP1:91,2] = PR[GP1:90,2] + -9.988;
   1:L PR[91] R[100]mm/sec CNT100;
   1:  PR[GP1:91,1] = PR[GP1:90,1] + 38.639;
   1:  PR[GP1:91,2] = PR[GP1:90,2] + -9.459;
   1:L PR[91] R[100]mm/sec CNT100;
   1:  PR[GP1:91,1] = PR[GP1:90,1] + 40.430;
   1:  PR[GP1:91,2] = PR[GP1:90,2] + -5.068;
   1:L PR[91] R[100]mm/sec CNT100;
   1:  PR[GP1:91,1] = PR[GP1:90,1] + 41.011;
   1:  PR[GP1:91,2] = PR[GP1:90,2] + -0.562;
   1:L PR[91] R[100]mm/sec CNT100;
   1:  PR[GP1:91,1] = PR[GP1:90,1] + 41.059;
   1:  PR[GP1:91,2] = PR[GP1:90,2] + -0.283;
   1:L PR[91] R[100]mm/sec CNT100;
   1:  PR[GP1:91,1] = PR[GP1:90,1] + 40.431;
   1:  PR[GP1:91,2] = PR[GP1:90,2] + 4.440;
   1:L PR[91] R[100]mm/sec CNT100;
   1:  PR[GP1:91,1] = PR[GP1:90,1] + 38.640;
   1:  PR[GP1:91,2] = PR[GP1:90,2] + 8.834;
   1:L PR[91] R[100]mm/sec CNT100;
   1:  PR[GP1:91,1] = PR[GP1:90,1] + 38.264;
   1:  PR[GP1:91,2] = PR[GP1:90,2] + 9.364;
   1:L PR[91] R[100]mm/sec CNT100;
   1:  PR[GP1:91,1] = PR[GP1:90,1] + 35.794;
   1:  PR[GP1:91,2] = PR[GP1:90,2] + 12.704;
   1:L PR[91] R[100]mm/sec CNT100;
   1:  PR[GP1:91,1] = PR[GP1:90,1] + 34.985;
   1:  PR[GP1:91,2] = PR[GP1:90,2] + 13.396;
   1:L PR[91] R[100]mm/sec CNT100;
   1:  PR[GP1:91,1] = PR[GP1:90,1] + 32.089;
   1:  PR[GP1:91,2] = PR[GP1:90,2] + 15.742;
   1:L PR[91] R[100]mm/sec CNT100;
   1:  PR[GP1:91,1] = PR[GP1:90,1] + 30.597;
   1:  PR[GP1:91,2] = PR[GP1:90,2] + 16.492;
   1:L PR[91] R[100]mm/sec CNT100;
   1:  PR[GP1:91,1] = PR[GP1:90,1] + 27.768;
   1:  PR[GP1:91,2] = PR[GP1:90,2] + 17.801;
   1:L PR[91] R[100]mm/sec CNT100;
   1:  PR[GP1:91,1] = PR[GP1:90,1] + 25.382;
   1:  PR[GP1:91,2] = PR[GP1:90,2] + 18.356;
   1:L PR[91] R[100]mm/sec CNT100;
   1:  PR[GP1:91,1] = PR[GP1:90,1] + 23.112;
   1:  PR[GP1:91,2] = PR[GP1:90,2] + 18.789;
   1:L PR[91] R[100]mm/sec CNT100;
   1:  PR[GP1:91,1] = PR[GP1:90,1] + 19.741;
   1:  PR[GP1:91,2] = PR[GP1:90,2] + 18.760;
   1:L PR[91] R[100]mm/sec CNT100;
   1:  PR[GP1:91,1] = PR[GP1:90,1] + 18.404;
   1:  PR[GP1:91,2] = PR[GP1:90,2] + 18.685;
   1:L PR[91] R[100]mm/sec CNT100;
   1:  PR[GP1:91,1] = PR[GP1:90,1] + 14.156;
   1:  PR[GP1:91,2] = PR[GP1:90,2] + 17.618;
   1:L PR[91] R[100]mm/sec CNT100;
   1:  PR[GP1:91,1] = PR[GP1:90,1] + 13.904;
   1:  PR[GP1:91,2] = PR[GP1:90,2] + 17.539;
   1:L PR[91] R[100]mm/sec CNT100;
   1:  PR[GP1:91,1] = PR[GP1:90,1] + 12.204;
   1:  PR[GP1:91,2] = PR[GP1:90,2] + 16.647;
   1:L PR[91] R[100]mm/sec CNT100;
   1:  PR[GP1:91,1] = PR[GP1:90,1] + 9.686;
   1:  PR[GP1:91,2] = PR[GP1:90,2] + 15.389;
   1:L PR[91] R[100]mm/sec CNT100;
   1:  PR[GP1:91,1] = PR[GP1:90,1] + 9.488;
   1:  PR[GP1:91,2] = PR[GP1:90,2] + 15.258;
   1:L PR[91] R[100]mm/sec CNT100;
   1:  PR[GP1:91,1] = PR[GP1:90,1] + 6.499;
   1:  PR[GP1:91,2] = PR[GP1:90,2] + 12.701;
   1:L PR[91] R[100]mm/sec CNT100;
   1:  PR[GP1:91,1] = PR[GP1:90,1] + 5.943;
   1:  PR[GP1:91,2] = PR[GP1:90,2] + 12.191;
   1:L PR[91] R[100]mm/sec CNT100;
   1:  PR[GP1:91,1] = PR[GP1:90,1] + 5.298;
   1:  PR[GP1:91,2] = PR[GP1:90,2] + 11.359;
   1:L PR[91] R[100]mm/sec CNT100;
   1:  PR[GP1:91,1] = PR[GP1:90,1] + 3.416;
   1:  PR[GP1:91,2] = PR[GP1:90,2] + 8.673;
   1:L PR[91] R[100]mm/sec CNT100;
   1:  PR[GP1:91,1] = PR[GP1:90,1] + 3.160;
   1:  PR[GP1:91,2] = PR[GP1:90,2] + 8.400;
   1:L PR[91] R[100]mm/sec CNT100;
   1:  PR[GP1:91,1] = PR[GP1:90,1] + 2.654;
   1:  PR[GP1:91,2] = PR[GP1:90,2] + 7.930;
   1:L PR[91] R[100]mm/sec CNT100;
   1:  PR[GP1:91,1] = PR[GP1:90,1] + 2.184;
   1:  PR[GP1:91,2] = PR[GP1:90,2] + 7.596;
   1:L PR[91] R[100]mm/sec CNT100;
   1:  PR[GP1:91,1] = PR[GP1:90,1] + 1.035;
   1:  PR[GP1:91,2] = PR[GP1:90,2] + 7.316;
   1:L PR[91] R[100]mm/sec CNT100;
   1:  PR[GP1:91,1] = PR[GP1:90,1] + -0.870;
   1:L PR[91] R[100]mm/sec CNT100;
   1:  ! -- Layer/Ebene 32 -- !;
   1:  PR[91] = PR[90];
   1:  PR[GP1:91,1] = PR[GP1:90,1] + -1.952;
   1:  PR[GP1:91,2] = PR[GP1:90,2] + 7.891;
   1:  PR[GP1:91,3] = PR[GP1:90,3] + 19.825;
   1:L PR[91] R[100]mm/sec CNT100;
   1:  PR[GP1:91,1] = PR[GP1:90,1] + -2.380;
   1:  PR[GP1:91,2] = PR[GP1:90,2] + 8.195;
   1:L PR[91] R[100]mm/sec CNT100;
   1:  PR[GP1:91,1] = PR[GP1:90,1] + -2.936;
   1:  PR[GP1:91,2] = PR[GP1:90,2] + 8.712;
   1:L PR[91] R[100]mm/sec CNT100;
   1:  PR[GP1:91,1] = PR[GP1:90,1] + -3.151;
   1:  PR[GP1:91,2] = PR[GP1:90,2] + 8.945;
   1:L PR[91] R[100]mm/sec CNT100;
   1:  PR[GP1:91,1] = PR[GP1:90,1] + -4.565;
   1:  PR[GP1:91,2] = PR[GP1:90,2] + 10.958;
   1:L PR[91] R[100]mm/sec CNT100;
   1:  PR[GP1:91,1] = PR[GP1:90,1] + -5.544;
   1:  PR[GP1:91,2] = PR[GP1:90,2] + 12.223;
   1:L PR[91] R[100]mm/sec CNT100;
   1:  PR[GP1:91,1] = PR[GP1:90,1] + -8.080;
   1:  PR[GP1:91,2] = PR[GP1:90,2] + 14.401;
   1:L PR[91] R[100]mm/sec CNT100;
   1:  PR[GP1:91,1] = PR[GP1:90,1] + -8.920;
   1:  PR[GP1:91,2] = PR[GP1:90,2] + 15.161;
   1:L PR[91] R[100]mm/sec CNT100;
   1:  PR[GP1:91,1] = PR[GP1:90,1] + -9.513;
   1:  PR[GP1:91,2] = PR[GP1:90,2] + 15.553;
   1:L PR[91] R[100]mm/sec CNT100;
   1:  PR[GP1:91,1] = PR[GP1:90,1] + -13.535;
   1:  PR[GP1:91,2] = PR[GP1:90,2] + 17.563;
   1:L PR[91] R[100]mm/sec CNT100;
   1:  PR[GP1:91,1] = PR[GP1:90,1] + -13.583;
   1:  PR[GP1:91,2] = PR[GP1:90,2] + 17.585;
   1:L PR[91] R[100]mm/sec CNT100;
   1:  PR[GP1:91,1] = PR[GP1:90,1] + -14.727;
   1:  PR[GP1:91,2] = PR[GP1:90,2] + 17.856;
   1:L PR[91] R[100]mm/sec CNT100;
   1:  PR[GP1:91,1] = PR[GP1:90,1] + -18.240;
   1:  PR[GP1:91,2] = PR[GP1:90,2] + 18.735;
   1:L PR[91] R[100]mm/sec CNT100;
   1:  PR[GP1:91,1] = PR[GP1:90,1] + -18.896;
   1:  PR[GP1:91,2] = PR[GP1:90,2] + 18.772;
   1:L PR[91] R[100]mm/sec CNT100;
   1:  PR[GP1:91,1] = PR[GP1:90,1] + -22.930;
   1:  PR[GP1:91,2] = PR[GP1:90,2] + 18.805;
   1:L PR[91] R[100]mm/sec CNT100;
   1:  PR[GP1:91,1] = PR[GP1:90,1] + -24.571;
   1:  PR[GP1:91,2] = PR[GP1:90,2] + 18.492;
   1:L PR[91] R[100]mm/sec CNT100;
   1:  PR[GP1:91,1] = PR[GP1:90,1] + -27.564;
   1:  PR[GP1:91,2] = PR[GP1:90,2] + 17.796;
   1:L PR[91] R[100]mm/sec CNT100;
   1:  PR[GP1:91,1] = PR[GP1:90,1] + -29.848;
   1:  PR[GP1:91,2] = PR[GP1:90,2] + 16.738;
   1:L PR[91] R[100]mm/sec CNT100;
   1:  PR[GP1:91,1] = PR[GP1:90,1] + -31.863;
   1:  PR[GP1:91,2] = PR[GP1:90,2] + 15.722;
   1:L PR[91] R[100]mm/sec CNT100;
   1:  PR[GP1:91,1] = PR[GP1:90,1] + -34.323;
   1:  PR[GP1:91,2] = PR[GP1:90,2] + 13.730;
   1:L PR[91] R[100]mm/sec CNT100;
   1:  PR[GP1:91,1] = PR[GP1:90,1] + -35.549;
   1:  PR[GP1:91,2] = PR[GP1:90,2] + 12.684;
   1:L PR[91] R[100]mm/sec CNT100;
   1:  PR[GP1:91,1] = PR[GP1:90,1] + -37.705;
   1:  PR[GP1:91,2] = PR[GP1:90,2] + 9.771;
   1:L PR[91] R[100]mm/sec CNT100;
   1:  PR[GP1:91,1] = PR[GP1:90,1] + -38.379;
   1:  PR[GP1:91,2] = PR[GP1:90,2] + 8.822;
   1:L PR[91] R[100]mm/sec CNT100;
   1:  PR[GP1:91,1] = PR[GP1:90,1] + -40.160;
   1:  PR[GP1:91,2] = PR[GP1:90,2] + 4.424;
   1:L PR[91] R[100]mm/sec CNT100;
   1:  PR[GP1:91,1] = PR[GP1:90,1] + -40.679;
   1:  PR[GP1:91,2] = PR[GP1:90,2] + 0.404;
   1:L PR[91] R[100]mm/sec CNT100;
   1:  PR[GP1:91,1] = PR[GP1:90,1] + -40.751;
   1:  PR[GP1:91,2] = PR[GP1:90,2] + -0.004;
   1:L PR[91] R[100]mm/sec CNT100;
   1:  PR[GP1:91,1] = PR[GP1:90,1] + -40.788;
   1:  PR[GP1:91,2] = PR[GP1:90,2] + -0.306;
   1:L PR[91] R[100]mm/sec CNT100;
   1:  PR[GP1:91,1] = PR[GP1:90,1] + -40.160;
   1:  PR[GP1:91,2] = PR[GP1:90,2] + -5.052;
   1:L PR[91] R[100]mm/sec CNT100;
   1:  PR[GP1:91,1] = PR[GP1:90,1] + -39.840;
   1:  PR[GP1:91,2] = PR[GP1:90,2] + -5.861;
   1:L PR[91] R[100]mm/sec CNT100;
   1:  PR[GP1:91,1] = PR[GP1:90,1] + -38.379;
   1:  PR[GP1:91,2] = PR[GP1:90,2] + -9.445;
   1:L PR[91] R[100]mm/sec CNT100;
   1:  PR[GP1:91,1] = PR[GP1:90,1] + -37.705;
   1:  PR[GP1:91,2] = PR[GP1:90,2] + -10.394;
   1:L PR[91] R[100]mm/sec CNT100;
   1:  PR[GP1:91,1] = PR[GP1:90,1] + -35.549;
   1:  PR[GP1:91,2] = PR[GP1:90,2] + -13.308;
   1:L PR[91] R[100]mm/sec CNT100;
   1:  PR[GP1:91,1] = PR[GP1:90,1] + -34.323;
   1:  PR[GP1:91,2] = PR[GP1:90,2] + -14.354;
   1:L PR[91] R[100]mm/sec CNT100;
   1:  PR[GP1:91,1] = PR[GP1:90,1] + -31.862;
   1:  PR[GP1:91,2] = PR[GP1:90,2] + -16.347;
   1:L PR[91] R[100]mm/sec CNT100;
   1:  PR[GP1:91,1] = PR[GP1:90,1] + -29.848;
   1:  PR[GP1:91,2] = PR[GP1:90,2] + -17.362;
   1:L PR[91] R[100]mm/sec CNT100;
   1:  PR[GP1:91,1] = PR[GP1:90,1] + -27.563;
   1:  PR[GP1:91,2] = PR[GP1:90,2] + -18.420;
   1:L PR[91] R[100]mm/sec CNT100;
   1:  PR[GP1:91,1] = PR[GP1:90,1] + -24.570;
   1:  PR[GP1:91,2] = PR[GP1:90,2] + -19.117;
   1:L PR[91] R[100]mm/sec CNT100;
   1:  PR[GP1:91,1] = PR[GP1:90,1] + -22.930;
   1:  PR[GP1:91,2] = PR[GP1:90,2] + -19.429;
   1:L PR[91] R[100]mm/sec CNT100;
   1:  PR[GP1:91,1] = PR[GP1:90,1] + -18.895;
   1:  PR[GP1:91,2] = PR[GP1:90,2] + -19.396;
   1:L PR[91] R[100]mm/sec CNT100;
   1:  PR[GP1:91,1] = PR[GP1:90,1] + -18.240;
   1:  PR[GP1:91,2] = PR[GP1:90,2] + -19.359;
   1:L PR[91] R[100]mm/sec CNT100;
   1:  PR[GP1:91,1] = PR[GP1:90,1] + -14.724;
   1:  PR[GP1:91,2] = PR[GP1:90,2] + -18.479;
   1:L PR[91] R[100]mm/sec CNT100;
   1:  PR[GP1:91,1] = PR[GP1:90,1] + -13.617;
   1:  PR[GP1:91,2] = PR[GP1:90,2] + -18.222;
   1:L PR[91] R[100]mm/sec CNT100;
   1:  PR[GP1:91,1] = PR[GP1:90,1] + -13.604;
   1:  PR[GP1:91,2] = PR[GP1:90,2] + -18.219;
   1:L PR[91] R[100]mm/sec CNT100;
   1:  PR[GP1:91,1] = PR[GP1:90,1] + -13.534;
   1:  PR[GP1:91,2] = PR[GP1:90,2] + -18.187;
   1:L PR[91] R[100]mm/sec CNT100;
   1:  PR[GP1:91,1] = PR[GP1:90,1] + -9.512;
   1:  PR[GP1:91,2] = PR[GP1:90,2] + -16.176;
   1:L PR[91] R[100]mm/sec CNT100;
   1:  PR[GP1:91,1] = PR[GP1:90,1] + -8.902;
   1:  PR[GP1:91,2] = PR[GP1:90,2] + -15.773;
   1:L PR[91] R[100]mm/sec CNT100;
   1:  PR[GP1:91,1] = PR[GP1:90,1] + -6.439;
   1:  PR[GP1:91,2] = PR[GP1:90,2] + -13.673;
   1:L PR[91] R[100]mm/sec CNT100;
   1:  PR[GP1:91,1] = PR[GP1:90,1] + -5.558;
   1:  PR[GP1:91,2] = PR[GP1:90,2] + -12.866;
   1:L PR[91] R[100]mm/sec CNT100;
   1:  PR[GP1:91,1] = PR[GP1:90,1] + -4.564;
   1:  PR[GP1:91,2] = PR[GP1:90,2] + -11.582;
   1:L PR[91] R[100]mm/sec CNT100;
   1:  PR[GP1:91,1] = PR[GP1:90,1] + -3.126;
   1:  PR[GP1:91,2] = PR[GP1:90,2] + -9.532;
   1:L PR[91] R[100]mm/sec CNT100;
   1:  PR[GP1:91,1] = PR[GP1:90,1] + -2.389;
   1:  PR[GP1:91,2] = PR[GP1:90,2] + -8.826;
   1:L PR[91] R[100]mm/sec CNT100;
   1:  PR[GP1:91,1] = PR[GP1:90,1] + -1.952;
   1:  PR[GP1:91,2] = PR[GP1:90,2] + -8.515;
   1:L PR[91] R[100]mm/sec CNT100;
   1:  PR[GP1:91,1] = PR[GP1:90,1] + -0.791;
   1:  PR[GP1:91,2] = PR[GP1:90,2] + -8.229;
   1:L PR[91] R[100]mm/sec CNT100;
   1:  PR[GP1:91,1] = PR[GP1:90,1] + 0.952;
   1:L PR[91] R[100]mm/sec CNT100;
   1:  PR[GP1:91,1] = PR[GP1:90,1] + 2.112;
   1:  PR[GP1:91,2] = PR[GP1:90,2] + -8.514;
   1:L PR[91] R[100]mm/sec CNT100;
   1:  PR[GP1:91,1] = PR[GP1:90,1] + 2.540;
   1:  PR[GP1:91,2] = PR[GP1:90,2] + -8.817;
   1:L PR[91] R[100]mm/sec CNT100;
   1:  PR[GP1:91,1] = PR[GP1:90,1] + 2.649;
   1:  PR[GP1:91,2] = PR[GP1:90,2] + -8.919;
   1:L PR[91] R[100]mm/sec CNT100;
   1:  PR[GP1:91,1] = PR[GP1:90,1] + 2.833;
   1:  PR[GP1:91,2] = PR[GP1:90,2] + -8.884;
   1:L PR[91] R[100]mm/sec CNT100;
   1:  PR[GP1:91,1] = PR[GP1:90,1] + 4.725;
   1:  PR[GP1:91,2] = PR[GP1:90,2] + -11.579;
   1:L PR[91] R[100]mm/sec CNT100;
   1:  PR[GP1:91,1] = PR[GP1:90,1] + 5.713;
   1:  PR[GP1:91,2] = PR[GP1:90,2] + -12.855;
   1:L PR[91] R[100]mm/sec CNT100;
   1:  PR[GP1:91,1] = PR[GP1:90,1] + 8.248;
   1:  PR[GP1:91,2] = PR[GP1:90,2] + -15.038;
   1:L PR[91] R[100]mm/sec CNT100;
   1:  PR[GP1:91,1] = PR[GP1:90,1] + 9.083;
   1:  PR[GP1:91,2] = PR[GP1:90,2] + -15.793;
   1:L PR[91] R[100]mm/sec CNT100;
   1:  PR[GP1:91,1] = PR[GP1:90,1] + 9.666;
   1:  PR[GP1:91,2] = PR[GP1:90,2] + -16.178;
   1:L PR[91] R[100]mm/sec CNT100;
   1:  PR[GP1:91,1] = PR[GP1:90,1] + 13.766;
   1:  PR[GP1:91,2] = PR[GP1:90,2] + -18.214;
   1:L PR[91] R[100]mm/sec CNT100;
   1:  PR[GP1:91,1] = PR[GP1:90,1] + 14.885;
   1:  PR[GP1:91,2] = PR[GP1:90,2] + -18.479;
   1:L PR[91] R[100]mm/sec CNT100;
   1:  PR[GP1:91,1] = PR[GP1:90,1] + 18.396;
   1:  PR[GP1:91,2] = PR[GP1:90,2] + -19.360;
   1:L PR[91] R[100]mm/sec CNT100;
   1:  PR[GP1:91,1] = PR[GP1:90,1] + 19.051;
   1:  PR[GP1:91,2] = PR[GP1:90,2] + -19.397;
   1:L PR[91] R[100]mm/sec CNT100;
   1:  PR[GP1:91,1] = PR[GP1:90,1] + 23.086;
   1:  PR[GP1:91,2] = PR[GP1:90,2] + -19.430;
   1:L PR[91] R[100]mm/sec CNT100;
   1:  PR[GP1:91,1] = PR[GP1:90,1] + 24.725;
   1:  PR[GP1:91,2] = PR[GP1:90,2] + -19.117;
   1:L PR[91] R[100]mm/sec CNT100;
   1:  PR[GP1:91,1] = PR[GP1:90,1] + 27.719;
   1:  PR[GP1:91,2] = PR[GP1:90,2] + -18.419;
   1:L PR[91] R[100]mm/sec CNT100;
   1:  PR[GP1:91,1] = PR[GP1:90,1] + 30.004;
   1:  PR[GP1:91,2] = PR[GP1:90,2] + -17.362;
   1:L PR[91] R[100]mm/sec CNT100;
   1:  PR[GP1:91,1] = PR[GP1:90,1] + 32.018;
   1:  PR[GP1:91,2] = PR[GP1:90,2] + -16.349;
   1:L PR[91] R[100]mm/sec CNT100;
   1:  PR[GP1:91,1] = PR[GP1:90,1] + 34.479;
   1:  PR[GP1:91,2] = PR[GP1:90,2] + -14.356;
   1:L PR[91] R[100]mm/sec CNT100;
   1:  PR[GP1:91,1] = PR[GP1:90,1] + 35.704;
   1:  PR[GP1:91,2] = PR[GP1:90,2] + -13.308;
   1:L PR[91] R[100]mm/sec CNT100;
   1:  PR[GP1:91,1] = PR[GP1:90,1] + 37.861;
   1:  PR[GP1:91,2] = PR[GP1:90,2] + -10.392;
   1:L PR[91] R[100]mm/sec CNT100;
   1:  PR[GP1:91,1] = PR[GP1:90,1] + 38.535;
   1:  PR[GP1:91,2] = PR[GP1:90,2] + -9.441;
   1:L PR[91] R[100]mm/sec CNT100;
   1:  PR[GP1:91,1] = PR[GP1:90,1] + 40.317;
   1:  PR[GP1:91,2] = PR[GP1:90,2] + -5.061;
   1:L PR[91] R[100]mm/sec CNT100;
   1:  PR[GP1:91,1] = PR[GP1:90,1] + 40.836;
   1:  PR[GP1:91,2] = PR[GP1:90,2] + -1.032;
   1:L PR[91] R[100]mm/sec CNT100;
   1:  PR[GP1:91,1] = PR[GP1:90,1] + 40.908;
   1:  PR[GP1:91,2] = PR[GP1:90,2] + -0.623;
   1:L PR[91] R[100]mm/sec CNT100;
   1:  PR[GP1:91,1] = PR[GP1:90,1] + 40.945;
   1:  PR[GP1:91,2] = PR[GP1:90,2] + -0.318;
   1:L PR[91] R[100]mm/sec CNT100;
   1:  PR[GP1:91,1] = PR[GP1:90,1] + 40.318;
   1:  PR[GP1:91,2] = PR[GP1:90,2] + 4.434;
   1:L PR[91] R[100]mm/sec CNT100;
   1:  PR[GP1:91,1] = PR[GP1:90,1] + 38.535;
   1:  PR[GP1:91,2] = PR[GP1:90,2] + 8.817;
   1:L PR[91] R[100]mm/sec CNT100;
   1:  PR[GP1:91,1] = PR[GP1:90,1] + 37.861;
   1:  PR[GP1:91,2] = PR[GP1:90,2] + 9.768;
   1:L PR[91] R[100]mm/sec CNT100;
   1:  PR[GP1:91,1] = PR[GP1:90,1] + 35.704;
   1:  PR[GP1:91,2] = PR[GP1:90,2] + 12.684;
   1:L PR[91] R[100]mm/sec CNT100;
   1:  PR[GP1:91,1] = PR[GP1:90,1] + 34.478;
   1:  PR[GP1:91,2] = PR[GP1:90,2] + 13.732;
   1:L PR[91] R[100]mm/sec CNT100;
   1:  PR[GP1:91,1] = PR[GP1:90,1] + 32.018;
   1:  PR[GP1:91,2] = PR[GP1:90,2] + 15.726;
   1:L PR[91] R[100]mm/sec CNT100;
   1:  PR[GP1:91,1] = PR[GP1:90,1] + 30.002;
   1:  PR[GP1:91,2] = PR[GP1:90,2] + 16.739;
   1:L PR[91] R[100]mm/sec CNT100;
   1:  PR[GP1:91,1] = PR[GP1:90,1] + 27.717;
   1:  PR[GP1:91,2] = PR[GP1:90,2] + 17.796;
   1:L PR[91] R[100]mm/sec CNT100;
   1:  PR[GP1:91,1] = PR[GP1:90,1] + 24.720;
   1:  PR[GP1:91,2] = PR[GP1:90,2] + 18.493;
   1:L PR[91] R[100]mm/sec CNT100;
   1:  PR[GP1:91,1] = PR[GP1:90,1] + 23.081;
   1:  PR[GP1:91,2] = PR[GP1:90,2] + 18.806;
   1:L PR[91] R[100]mm/sec CNT100;
   1:  PR[GP1:91,1] = PR[GP1:90,1] + 19.042;
   1:  PR[GP1:91,2] = PR[GP1:90,2] + 18.771;
   1:L PR[91] R[100]mm/sec CNT100;
   1:  PR[GP1:91,1] = PR[GP1:90,1] + 18.389;
   1:  PR[GP1:91,2] = PR[GP1:90,2] + 18.735;
   1:L PR[91] R[100]mm/sec CNT100;
   1:  PR[GP1:91,1] = PR[GP1:90,1] + 14.885;
   1:  PR[GP1:91,2] = PR[GP1:90,2] + 17.855;
   1:L PR[91] R[100]mm/sec CNT100;
   1:  PR[GP1:91,1] = PR[GP1:90,1] + 13.756;
   1:  PR[GP1:91,2] = PR[GP1:90,2] + 17.586;
   1:L PR[91] R[100]mm/sec CNT100;
   1:  PR[GP1:91,1] = PR[GP1:90,1] + 9.659;
   1:  PR[GP1:91,2] = PR[GP1:90,2] + 15.549;
   1:L PR[91] R[100]mm/sec CNT100;
   1:  PR[GP1:91,1] = PR[GP1:90,1] + 9.058;
   1:  PR[GP1:91,2] = PR[GP1:90,2] + 15.152;
   1:L PR[91] R[100]mm/sec CNT100;
   1:  PR[GP1:91,1] = PR[GP1:90,1] + 6.599;
   1:  PR[GP1:91,2] = PR[GP1:90,2] + 13.048;
   1:L PR[91] R[100]mm/sec CNT100;
   1:  PR[GP1:91,1] = PR[GP1:90,1] + 5.722;
   1:  PR[GP1:91,2] = PR[GP1:90,2] + 12.244;
   1:L PR[91] R[100]mm/sec CNT100;
   1:  PR[GP1:91,1] = PR[GP1:90,1] + 4.720;
   1:  PR[GP1:91,2] = PR[GP1:90,2] + 10.950;
   1:L PR[91] R[100]mm/sec CNT100;
   1:  PR[GP1:91,1] = PR[GP1:90,1] + 3.286;
   1:  PR[GP1:91,2] = PR[GP1:90,2] + 8.905;
   1:L PR[91] R[100]mm/sec CNT100;
   1:  PR[GP1:91,1] = PR[GP1:90,1] + 2.550;
   1:  PR[GP1:91,2] = PR[GP1:90,2] + 8.201;
   1:L PR[91] R[100]mm/sec CNT100;
   1:  PR[GP1:91,1] = PR[GP1:90,1] + 2.114;
   1:  PR[GP1:91,2] = PR[GP1:90,2] + 7.890;
   1:L PR[91] R[100]mm/sec CNT100;
   1:  PR[GP1:91,1] = PR[GP1:90,1] + 0.955;
   1:  PR[GP1:91,2] = PR[GP1:90,2] + 7.605;
   1:L PR[91] R[100]mm/sec CNT100;
   1:  PR[GP1:91,1] = PR[GP1:90,1] + -0.790;
   1:L PR[91] R[100]mm/sec CNT100;
   1:  ! -- Layer/Ebene 33 -- !;
   1:  PR[91] = PR[90];
   1:  PR[GP1:91,1] = PR[GP1:90,1] + -1.882;
   1:  PR[GP1:91,2] = PR[GP1:90,2] + 8.185;
   1:  PR[GP1:91,3] = PR[GP1:90,3] + 20.435;
   1:L PR[91] R[100]mm/sec CNT100;
   1:  PR[GP1:91,1] = PR[GP1:90,1] + -2.267;
   1:  PR[GP1:91,2] = PR[GP1:90,2] + 8.459;
   1:L PR[91] R[100]mm/sec CNT100;
   1:  PR[GP1:91,1] = PR[GP1:90,1] + -2.868;
   1:  PR[GP1:91,2] = PR[GP1:90,2] + 9.018;
   1:L PR[91] R[100]mm/sec CNT100;
   1:  PR[GP1:91,1] = PR[GP1:90,1] + -3.044;
   1:  PR[GP1:91,2] = PR[GP1:90,2] + 9.209;
   1:L PR[91] R[100]mm/sec CNT100;
   1:  PR[GP1:91,1] = PR[GP1:90,1] + -3.983;
   1:  PR[GP1:91,2] = PR[GP1:90,2] + 10.546;
   1:L PR[91] R[100]mm/sec CNT100;
   1:  PR[GP1:91,1] = PR[GP1:90,1] + -5.317;
   1:  PR[GP1:91,2] = PR[GP1:90,2] + 12.270;
   1:L PR[91] R[100]mm/sec CNT100;
   1:  PR[GP1:91,1] = PR[GP1:90,1] + -7.154;
   1:  PR[GP1:91,2] = PR[GP1:90,2] + 13.847;
   1:L PR[91] R[100]mm/sec CNT100;
   1:  PR[GP1:91,1] = PR[GP1:90,1] + -8.484;
   1:  PR[GP1:91,2] = PR[GP1:90,2] + 15.050;
   1:L PR[91] R[100]mm/sec CNT100;
   1:  PR[GP1:91,1] = PR[GP1:90,1] + -9.485;
   1:  PR[GP1:91,2] = PR[GP1:90,2] + 15.712;
   1:L PR[91] R[100]mm/sec CNT100;
   1:  PR[GP1:91,1] = PR[GP1:90,1] + -12.819;
   1:  PR[GP1:91,2] = PR[GP1:90,2] + 17.379;
   1:L PR[91] R[100]mm/sec CNT100;
   1:  PR[GP1:91,1] = PR[GP1:90,1] + -13.375;
   1:  PR[GP1:91,2] = PR[GP1:90,2] + 17.630;
   1:L PR[91] R[100]mm/sec CNT100;
   1:  PR[GP1:91,1] = PR[GP1:90,1] + -18.185;
   1:  PR[GP1:91,2] = PR[GP1:90,2] + 18.777;
   1:L PR[91] R[100]mm/sec CNT100;
   1:  PR[GP1:91,1] = PR[GP1:90,1] + -22.901;
   1:  PR[GP1:91,2] = PR[GP1:90,2] + 18.821;
   1:L PR[91] R[100]mm/sec CNT100;
   1:  PR[GP1:91,1] = PR[GP1:90,1] + -23.910;
   1:  PR[GP1:91,2] = PR[GP1:90,2] + 18.629;
   1:L PR[91] R[100]mm/sec CNT100;
   1:  PR[GP1:91,1] = PR[GP1:90,1] + -27.514;
   1:  PR[GP1:91,2] = PR[GP1:90,2] + 17.790;
   1:L PR[91] R[100]mm/sec CNT100;
   1:  PR[GP1:91,1] = PR[GP1:90,1] + -29.254;
   1:  PR[GP1:91,2] = PR[GP1:90,2] + 16.984;
   1:L PR[91] R[100]mm/sec CNT100;
   1:  PR[GP1:91,1] = PR[GP1:90,1] + -31.792;
   1:  PR[GP1:91,2] = PR[GP1:90,2] + 15.705;
   1:L PR[91] R[100]mm/sec CNT100;
   1:  PR[GP1:91,1] = PR[GP1:90,1] + -33.818;
   1:  PR[GP1:91,2] = PR[GP1:90,2] + 14.065;
   1:L PR[91] R[100]mm/sec CNT100;
   1:  PR[GP1:91,1] = PR[GP1:90,1] + -35.459;
   1:  PR[GP1:91,2] = PR[GP1:90,2] + 12.664;
   1:L PR[91] R[100]mm/sec CNT100;
   1:  PR[GP1:91,1] = PR[GP1:90,1] + -37.302;
   1:  PR[GP1:91,2] = PR[GP1:90,2] + 10.174;
   1:L PR[91] R[100]mm/sec CNT100;
   1:  PR[GP1:91,1] = PR[GP1:90,1] + -38.275;
   1:  PR[GP1:91,2] = PR[GP1:90,2] + 8.802;
   1:L PR[91] R[100]mm/sec CNT100;
   1:  PR[GP1:91,1] = PR[GP1:90,1] + -39.550;
   1:  PR[GP1:91,2] = PR[GP1:90,2] + 5.676;
   1:L PR[91] R[100]mm/sec CNT100;
   1:  PR[GP1:91,1] = PR[GP1:90,1] + -40.047;
   1:  PR[GP1:91,2] = PR[GP1:90,2] + 4.420;
   1:L PR[91] R[100]mm/sec CNT100;
   1:  PR[GP1:91,1] = PR[GP1:90,1] + -40.668;
   1:  PR[GP1:91,2] = PR[GP1:90,2] + -0.310;
   1:L PR[91] R[100]mm/sec CNT100;
   1:  PR[GP1:91,1] = PR[GP1:90,1] + -40.197;
   1:  PR[GP1:91,2] = PR[GP1:90,2] + -3.815;
   1:L PR[91] R[100]mm/sec CNT100;
   1:  PR[GP1:91,1] = PR[GP1:90,1] + -40.045;
   1:  PR[GP1:91,2] = PR[GP1:90,2] + -5.050;
   1:L PR[91] R[100]mm/sec CNT100;
   1:  PR[GP1:91,1] = PR[GP1:90,1] + -39.549;
   1:  PR[GP1:91,2] = PR[GP1:90,2] + -6.302;
   1:L PR[91] R[100]mm/sec CNT100;
   1:  PR[GP1:91,1] = PR[GP1:90,1] + -38.275;
   1:  PR[GP1:91,2] = PR[GP1:90,2] + -9.426;
   1:L PR[91] R[100]mm/sec CNT100;
   1:  PR[GP1:91,1] = PR[GP1:90,1] + -37.302;
   1:  PR[GP1:91,2] = PR[GP1:90,2] + -10.798;
   1:L PR[91] R[100]mm/sec CNT100;
   1:  PR[GP1:91,1] = PR[GP1:90,1] + -35.459;
   1:  PR[GP1:91,2] = PR[GP1:90,2] + -13.288;
   1:L PR[91] R[100]mm/sec CNT100;
   1:  PR[GP1:91,1] = PR[GP1:90,1] + -33.817;
   1:  PR[GP1:91,2] = PR[GP1:90,2] + -14.689;
   1:L PR[91] R[100]mm/sec CNT100;
   1:  PR[GP1:91,1] = PR[GP1:90,1] + -31.791;
   1:  PR[GP1:91,2] = PR[GP1:90,2] + -16.330;
   1:L PR[91] R[100]mm/sec CNT100;
   1:  PR[GP1:91,1] = PR[GP1:90,1] + -29.253;
   1:  PR[GP1:91,2] = PR[GP1:90,2] + -17.608;
   1:L PR[91] R[100]mm/sec CNT100;
   1:  PR[GP1:91,1] = PR[GP1:90,1] + -27.513;
   1:  PR[GP1:91,2] = PR[GP1:90,2] + -18.415;
   1:L PR[91] R[100]mm/sec CNT100;
   1:  PR[GP1:91,1] = PR[GP1:90,1] + -23.910;
   1:  PR[GP1:91,2] = PR[GP1:90,2] + -19.253;
   1:L PR[91] R[100]mm/sec CNT100;
   1:  PR[GP1:91,1] = PR[GP1:90,1] + -22.901;
   1:  PR[GP1:91,2] = PR[GP1:90,2] + -19.445;
   1:L PR[91] R[100]mm/sec CNT100;
   1:  PR[GP1:91,1] = PR[GP1:90,1] + -18.182;
   1:  PR[GP1:91,2] = PR[GP1:90,2] + -19.401;
   1:L PR[91] R[100]mm/sec CNT100;
   1:  PR[GP1:91,1] = PR[GP1:90,1] + -13.786;
   1:  PR[GP1:91,2] = PR[GP1:90,2] + -18.369;
   1:L PR[91] R[100]mm/sec CNT100;
   1:  PR[GP1:91,1] = PR[GP1:90,1] + -13.395;
   1:  PR[GP1:91,2] = PR[GP1:90,2] + -18.263;
   1:L PR[91] R[100]mm/sec CNT100;
   1:  PR[GP1:91,1] = PR[GP1:90,1] + -12.818;
   1:  PR[GP1:91,2] = PR[GP1:90,2] + -18.003;
   1:L PR[91] R[100]mm/sec CNT100;
   1:  PR[GP1:91,1] = PR[GP1:90,1] + -9.485;
   1:  PR[GP1:91,2] = PR[GP1:90,2] + -16.336;
   1:L PR[91] R[100]mm/sec CNT100;
   1:  PR[GP1:91,1] = PR[GP1:90,1] + -8.466;
   1:  PR[GP1:91,2] = PR[GP1:90,2] + -15.662;
   1:L PR[91] R[100]mm/sec CNT100;
   1:  PR[GP1:91,1] = PR[GP1:90,1] + -6.535;
   1:  PR[GP1:91,2] = PR[GP1:90,2] + -14.016;
   1:L PR[91] R[100]mm/sec CNT100;
   1:  PR[GP1:91,1] = PR[GP1:90,1] + -5.332;
   1:  PR[GP1:91,2] = PR[GP1:90,2] + -12.912;
   1:L PR[91] R[100]mm/sec CNT100;
   1:  PR[GP1:91,1] = PR[GP1:90,1] + -3.983;
   1:  PR[GP1:91,2] = PR[GP1:90,2] + -11.170;
   1:L PR[91] R[100]mm/sec CNT100;
   1:  PR[GP1:91,1] = PR[GP1:90,1] + -3.016;
   1:  PR[GP1:91,2] = PR[GP1:90,2] + -9.793;
   1:L PR[91] R[100]mm/sec CNT100;
   1:  PR[GP1:91,1] = PR[GP1:90,1] + -2.273;
   1:  PR[GP1:91,2] = PR[GP1:90,2] + -9.087;
   1:L PR[91] R[100]mm/sec CNT100;
   1:  PR[GP1:91,1] = PR[GP1:90,1] + -1.881;
   1:  PR[GP1:91,2] = PR[GP1:90,2] + -8.809;
   1:L PR[91] R[100]mm/sec CNT100;
   1:  PR[GP1:91,1] = PR[GP1:90,1] + -0.711;
   1:  PR[GP1:91,2] = PR[GP1:90,2] + -8.517;
   1:L PR[91] R[100]mm/sec CNT100;
   1:  PR[GP1:91,1] = PR[GP1:90,1] + 0.873;
   1:L PR[91] R[100]mm/sec CNT100;
   1:  PR[GP1:91,1] = PR[GP1:90,1] + 2.042;
   1:  PR[GP1:91,2] = PR[GP1:90,2] + -8.808;
   1:L PR[91] R[100]mm/sec CNT100;
   1:  PR[GP1:91,1] = PR[GP1:90,1] + 2.427;
   1:  PR[GP1:91,2] = PR[GP1:90,2] + -9.081;
   1:L PR[91] R[100]mm/sec CNT100;
   1:  PR[GP1:91,1] = PR[GP1:90,1] + 2.538;
   1:  PR[GP1:91,2] = PR[GP1:90,2] + -9.184;
   1:L PR[91] R[100]mm/sec CNT100;
   1:  PR[GP1:91,1] = PR[GP1:90,1] + 2.727;
   1:  PR[GP1:91,2] = PR[GP1:90,2] + -9.149;
   1:L PR[91] R[100]mm/sec CNT100;
   1:  PR[GP1:91,1] = PR[GP1:90,1] + 4.145;
   1:  PR[GP1:91,2] = PR[GP1:90,2] + -11.168;
   1:L PR[91] R[100]mm/sec CNT100;
   1:  PR[GP1:91,1] = PR[GP1:90,1] + 5.491;
   1:  PR[GP1:91,2] = PR[GP1:90,2] + -12.907;
   1:L PR[91] R[100]mm/sec CNT100;
   1:  PR[GP1:91,1] = PR[GP1:90,1] + 7.329;
   1:  PR[GP1:91,2] = PR[GP1:90,2] + -14.489;
   1:L PR[91] R[100]mm/sec CNT100;
   1:  PR[GP1:91,1] = PR[GP1:90,1] + 8.651;
   1:  PR[GP1:91,2] = PR[GP1:90,2] + -15.685;
   1:L PR[91] R[100]mm/sec CNT100;
   1:  PR[GP1:91,1] = PR[GP1:90,1] + 9.640;
   1:  PR[GP1:91,2] = PR[GP1:90,2] + -16.338;
   1:L PR[91] R[100]mm/sec CNT100;
   1:  PR[GP1:91,1] = PR[GP1:90,1] + 12.973;
   1:  PR[GP1:91,2] = PR[GP1:90,2] + -18.001;
   1:L PR[91] R[100]mm/sec CNT100;
   1:  PR[GP1:91,1] = PR[GP1:90,1] + 13.529;
   1:  PR[GP1:91,2] = PR[GP1:90,2] + -18.251;
   1:L PR[91] R[100]mm/sec CNT100;
   1:  PR[GP1:91,1] = PR[GP1:90,1] + 18.342;
   1:  PR[GP1:91,2] = PR[GP1:90,2] + -19.401;
   1:L PR[91] R[100]mm/sec CNT100;
   1:  PR[GP1:91,1] = PR[GP1:90,1] + 23.057;
   1:  PR[GP1:91,2] = PR[GP1:90,2] + -19.446;
   1:L PR[91] R[100]mm/sec CNT100;
   1:  PR[GP1:91,1] = PR[GP1:90,1] + 24.066;
   1:  PR[GP1:91,2] = PR[GP1:90,2] + -19.254;
   1:L PR[91] R[100]mm/sec CNT100;
   1:  PR[GP1:91,1] = PR[GP1:90,1] + 27.669;
   1:  PR[GP1:91,2] = PR[GP1:90,2] + -18.413;
   1:L PR[91] R[100]mm/sec CNT100;
   1:  PR[GP1:91,1] = PR[GP1:90,1] + 29.410;
   1:  PR[GP1:91,2] = PR[GP1:90,2] + -17.608;
   1:L PR[91] R[100]mm/sec CNT100;
   1:  PR[GP1:91,1] = PR[GP1:90,1] + 31.947;
   1:  PR[GP1:91,2] = PR[GP1:90,2] + -16.332;
   1:L PR[91] R[100]mm/sec CNT100;
   1:  PR[GP1:91,1] = PR[GP1:90,1] + 33.973;
   1:  PR[GP1:91,2] = PR[GP1:90,2] + -14.691;
   1:L PR[91] R[100]mm/sec CNT100;
   1:  PR[GP1:91,1] = PR[GP1:90,1] + 35.615;
   1:  PR[GP1:91,2] = PR[GP1:90,2] + -13.288;
   1:L PR[91] R[100]mm/sec CNT100;
   1:  PR[GP1:91,1] = PR[GP1:90,1] + 37.458;
   1:  PR[GP1:91,2] = PR[GP1:90,2] + -10.795;
   1:L PR[91] R[100]mm/sec CNT100;
   1:  PR[GP1:91,1] = PR[GP1:90,1] + 38.431;
   1:  PR[GP1:91,2] = PR[GP1:90,2] + -9.424;
   1:L PR[91] R[100]mm/sec CNT100;
   1:  PR[GP1:91,1] = PR[GP1:90,1] + 40.204;
   1:  PR[GP1:91,2] = PR[GP1:90,2] + -5.052;
   1:L PR[91] R[100]mm/sec CNT100;
   1:  PR[GP1:91,1] = PR[GP1:90,1] + 40.825;
   1:  PR[GP1:91,2] = PR[GP1:90,2] + -0.314;
   1:L PR[91] R[100]mm/sec CNT100;
   1:  PR[GP1:91,1] = PR[GP1:90,1] + 40.354;
   1:  PR[GP1:91,2] = PR[GP1:90,2] + 3.200;
   1:L PR[91] R[100]mm/sec CNT100;
   1:  PR[GP1:91,1] = PR[GP1:90,1] + 40.202;
   1:  PR[GP1:91,2] = PR[GP1:90,2] + 4.434;
   1:L PR[91] R[100]mm/sec CNT100;
   1:  PR[GP1:91,1] = PR[GP1:90,1] + 38.431;
   1:  PR[GP1:91,2] = PR[GP1:90,2] + 8.799;
   1:L PR[91] R[100]mm/sec CNT100;
   1:  PR[GP1:91,1] = PR[GP1:90,1] + 37.458;
   1:  PR[GP1:91,2] = PR[GP1:90,2] + 10.172;
   1:L PR[91] R[100]mm/sec CNT100;
   1:  PR[GP1:91,1] = PR[GP1:90,1] + 35.615;
   1:  PR[GP1:91,2] = PR[GP1:90,2] + 12.664;
   1:L PR[91] R[100]mm/sec CNT100;
   1:  PR[GP1:91,1] = PR[GP1:90,1] + 33.971;
   1:  PR[GP1:91,2] = PR[GP1:90,2] + 14.068;
   1:L PR[91] R[100]mm/sec CNT100;
   1:  PR[GP1:91,1] = PR[GP1:90,1] + 31.946;
   1:  PR[GP1:91,2] = PR[GP1:90,2] + 15.709;
   1:L PR[91] R[100]mm/sec CNT100;
   1:  PR[GP1:91,1] = PR[GP1:90,1] + 29.407;
   1:  PR[GP1:91,2] = PR[GP1:90,2] + 16.985;
   1:L PR[91] R[100]mm/sec CNT100;
   1:  PR[GP1:91,1] = PR[GP1:90,1] + 27.666;
   1:  PR[GP1:91,2] = PR[GP1:90,2] + 17.790;
   1:L PR[91] R[100]mm/sec CNT100;
   1:  PR[GP1:91,1] = PR[GP1:90,1] + 24.059;
   1:  PR[GP1:91,2] = PR[GP1:90,2] + 18.630;
   1:L PR[91] R[100]mm/sec CNT100;
   1:  PR[GP1:91,1] = PR[GP1:90,1] + 23.050;
   1:  PR[GP1:91,2] = PR[GP1:90,2] + 18.823;
   1:L PR[91] R[100]mm/sec CNT100;
   1:  PR[GP1:91,1] = PR[GP1:90,1] + 18.358;
   1:  PR[GP1:91,2] = PR[GP1:90,2] + 18.783;
   1:L PR[91] R[100]mm/sec CNT100;
   1:  PR[GP1:91,1] = PR[GP1:90,1] + 13.935;
   1:  PR[GP1:91,2] = PR[GP1:90,2] + 17.740;
   1:L PR[91] R[100]mm/sec CNT100;
   1:  PR[GP1:91,1] = PR[GP1:90,1] + 13.541;
   1:  PR[GP1:91,2] = PR[GP1:90,2] + 17.633;
   1:L PR[91] R[100]mm/sec CNT100;
   1:  PR[GP1:91,1] = PR[GP1:90,1] + 12.963;
   1:  PR[GP1:91,2] = PR[GP1:90,2] + 17.373;
   1:L PR[91] R[100]mm/sec CNT100;
   1:  PR[GP1:91,1] = PR[GP1:90,1] + 9.633;
   1:  PR[GP1:91,2] = PR[GP1:90,2] + 15.710;
   1:L PR[91] R[100]mm/sec CNT100;
   1:  PR[GP1:91,1] = PR[GP1:90,1] + 8.628;
   1:  PR[GP1:91,2] = PR[GP1:90,2] + 15.046;
   1:L PR[91] R[100]mm/sec CNT100;
   1:  PR[GP1:91,1] = PR[GP1:90,1] + 6.699;
   1:  PR[GP1:91,2] = PR[GP1:90,2] + 13.395;
   1:L PR[91] R[100]mm/sec CNT100;
   1:  PR[GP1:91,1] = PR[GP1:90,1] + 5.501;
   1:  PR[GP1:91,2] = PR[GP1:90,2] + 12.296;
   1:L PR[91] R[100]mm/sec CNT100;
   1:  PR[GP1:91,1] = PR[GP1:90,1] + 4.141;
   1:  PR[GP1:91,2] = PR[GP1:90,2] + 10.541;
   1:L PR[91] R[100]mm/sec CNT100;
   1:  PR[GP1:91,1] = PR[GP1:90,1] + 3.178;
   1:  PR[GP1:91,2] = PR[GP1:90,2] + 9.166;
   1:L PR[91] R[100]mm/sec CNT100;
   1:  PR[GP1:91,1] = PR[GP1:90,1] + 2.434;
   1:  PR[GP1:91,2] = PR[GP1:90,2] + 8.463;
   1:L PR[91] R[100]mm/sec CNT100;
   1:  PR[GP1:91,1] = PR[GP1:90,1] + 2.044;
   1:  PR[GP1:91,2] = PR[GP1:90,2] + 8.185;
   1:L PR[91] R[100]mm/sec CNT100;
   1:  PR[GP1:91,1] = PR[GP1:90,1] + 0.875;
   1:  PR[GP1:91,2] = PR[GP1:90,2] + 7.893;
   1:L PR[91] R[100]mm/sec CNT100;
   1:  PR[GP1:91,1] = PR[GP1:90,1] + -0.710;
   1:L PR[91] R[100]mm/sec CNT100 TB   .50sec,CALL END_PUD;
   1:  DO[117:Laser Start]=OFF;
   1:  !Sicherheitspunkt!;
   1:  PR[92] = PR[91];
   1:  PR[92] = PR[GP1:92,3] + 50;
   1:J PR[92];
   1:  WAIT   5.00(sec);
   1:  DO[119:Gas]=OFF;
   1:  CALL HOME_ALL;
/POS
/END
